// TwinCAT 3 PLC project motion
// Title: LCLS_OMotion
// Company: SLAC
// ProjectVersion: 6.0.0
// ProgramVersion: 3.1.4026.17
// libraries:
//   LCLS General, * (SLAC)
//   Tc2_EtherCAT, * (Beckhoff Automation GmbH)
//   Tc2_MC2, * (Beckhoff Automation GmbH)
//   Tc2_Standard, * (Beckhoff Automation GmbH)
//   Tc2_System, * (Beckhoff Automation GmbH)
//   Tc2_Utilities, * (Beckhoff Automation GmbH)
//   TcUnit, * (www.tcunit.org)
// project tree:
//   / DemoTask.TcTTO (not stored), PlcTask.TcTTO, UnitTestTask.TcTTO
//   DUTs/ E_LCLSMotionError.TcDUT, E_MotionLogLevel.TcDUT (not stored), MOTION_LOGGER_MSG.TcDUT (not stored), ST_ExtendedMotionStatus.TcDUT, E_HomeStates.TcDUT (not stored), E_Module.TcDUT (not stored), ST_MotionStatus.TcDUT, ENUM_StageEnableMode.TcDUT (not stored), E_DS402HomingMethod.TcDUT (not stored), E_DS402OpMode.TcDUT (not stored), E_EpicsHomeCmd.TcDUT, E_EpicsMotorCmd.TcDUT (not stored), E_MoveMode.TcDUT (not stored), E_MoveState.TcDUT, E_StageBrakeMode.TcDUT (not stored), E_StageEnableMode.TcDUT (not stored), ST_AxisParameterSetExposed.TcDUT (not stored), ST_DS402Drive.TcDUT, ST_DS402DriveStatus.TcDUT (not stored), ST_AxisStatus.TcDUT, ST_MotionCommand.TcDUT, ST_MotionLogMessage.TcDUT (not stored), ST_MoveRequestStatus.TcDUT
//   POUs/FBs/Common/ FB_EncoderScaling.TcPOU (not stored), FB_EpicsMotionParamsStatus.TcPOU (not stored), FB_EpicsMoveRequest.TcPOU (not stored), FB_LimSwStatus.TcPOU, FB_MotionDrive.TcPOU, FB_MotionDriveStateMachine.TcPOU (not stored), FB_MotionInterlocksCommon.TcPOU, FB_MotionInterlocksLimSw.TcPOU (not stored), FB_MotionLogger.TcPOU (not stored), FB_PersistentDataStorage.TcPOU (not stored)
//   POUs/FBs/Containers/ FB_MotionStageNC.TcPOU (not stored)
//   POUs/FBs/DS402/ FB_HomeDS402.TcPOU (excluded from build)
//   POUs/FBs/NC/ FB_AxisStatusNC.TcPOU (excluded from build), FB_BacklashCompensationNC.TcPOU, FB_BrakeNC.TcPOU, FB_HaltNC.TcPOU, FB_HomeNC.TcPOU, FB_MotionAxisNC.TcPOU, FB_MoveAbsoluteNC.TcPOU, FB_ParamsSaveRestoreNC.TcPOU, FB_PowerInterlockNC.TcPOU (not stored), FB_PowerNC.TcPOU, FB_ReadParameterNC.TcPOU, FB_ResetNC.TcPOU, FB_WriteParameterNC.TcPOU
//   POUs/ITFs/ I_AxisStatus.TcIO, I_BacklashCompensation.TcIO, I_Brake.TcIO, I_DS402GenericDrive.TcIO (not stored), I_EncoderScaling.TcIO (not stored), I_EpicsMotionParamsStatus.TcIO (not stored), I_Error.TcIO (not stored), I_Halt.TcIO, I_Home.TcIO, I_HomeDS402.TcIO (not stored), I_LimSwStatus.TcIO, I_MotionAxis.TcIO, I_MotionAxisDS402.TcIO, I_MotionDrive.TcIO, I_MotionInterlocks.TcIO, I_MotionInterlocksCommon.TcIO (not stored), I_MotionLogger.TcIO (not stored), I_MotionStage.TcIO (not stored), I_MoveAbsolute.TcIO, I_MoveRequest.TcIO (not stored), I_ParamsSaveRestore.TcIO (not stored), I_PersistentDataStorage.TcIO (not stored), I_Power.TcIO, I_ReadParameter.TcIO, I_Reset.TcIO, I_StateMachine.TcIO (not stored), I_Status.TcIO (not stored), I_StatusEx.TcIO (not stored), I_WriteParameter.TcIO (not stored)
//   Test/Containers/ FB_MotionStageNC_Test.TcPOU
//   Test/Interlok/ FB_MotionInterlocksCommon_Test.TcPOU, FB_MotionInterlocksLimSw_Test.TcPOU
//   Test/ HARD_TEST.TcPOU, PRG_TEST.TcPOU, CONTAINER_TEST.TcPOU
//   Test/Orchetration/ FB_BrakeNC_Test.TcPOU (not stored), FB_MotionDriveStateMachine_Test.TcPOU, FB_MotionDrive_Test.TcPOU, FB_MoveRequest_Test.TcPOU
//   Test/NC/ FB_NcMotionBlocks_Test.TcPOU, FB_MotionAxisNC_Test.TcPOU
//   Test/TestDouble/ FB_AxisStatusNC_TestDouble.TcPOU, FB_BacklashCompensationNC_TestDouble.TcPOU, FB_Brake_TestDouble.TcPOU (not stored), FB_EncoderScalingNC_TestDouble.TcPOU (not stored), FB_EpicsMotionParamsStatus_TestDouble.TcPOU, FB_HaltNC_TestDouble.TcPOU, FB_HomeNC_TestDouble.TcPOU, FB_LimSwStatus_testDouble.TcPOU, FB_MotionAxisDS402_TestDouble.TcPOU, FB_MotionAxisNC_TestDouble.TcPOU, FB_StateMachine_TestDouble.TcPOU, FB_MotionInterlocksCommon_TestDouble.TcPOU, FB_MotionInterlocksLimSw_TestDouble.TcPOU, FB_MotionLogger_TestDouble.TcPOU, FB_MoveAbsoluteNC_TestDouble.TcPOU, FB_MoveRequest_TestDouble.TcPOU, FB_ParamSaveRestoreNC_TestDouble.TcPOU (not stored), FB_PersistentDataStorage_TestDouble.TcPOU (not stored), FB_PowerNC_TestDouble.TcPOU, FB_ReadParameterNC_TestDouble.TcPOU (not stored), FB_ResetNC_TestDouble.TcPOU, FB_WriteParameterNC_TestDouble.TcPOU
//   Test/Utils/ FB_MotionLogger_Test.TcPOU
//   VISUs/ motion.TcCD (not stored)
// real-time tasks:
//   TASK PlcTask: cycle T#10ms, priority 1, ADS port 350
//   TASK UnitTestTask: cycle T#10ms, priority 20, ADS port 351
//   TASK Demo: cycle T#10ms, priority 2, ADS port 352
// motion (NC):
//   TASK NC-Task 1 SAF: cycle T#2ms, priority 4, ADS port 501
//   TASK NC-Task 1 SVB: cycle T#10ms, priority 8, ADS port 511
//   AXIS Axis_HomeNC_Test8 (id 15)
//     OtherSettings: AllowMotionCmdToSlave=true
//     encoder EncType=1
//     drive DrvType=5
//       Analog: TorqueSetpointScale=10, ScaleFactorActTorque=0.1
//       TimeComp: TaskDelayCycles=1
//     controller CtrType=1
//       CtrPara: PriorControlFactor=1
//         Observer: BandWidth=20
//   AXIS Axis_HomeNC_Test7 (id 14)
//     OtherSettings: AllowMotionCmdToSlave=true
//     encoder EncType=1
//     drive DrvType=5
//       Analog: TorqueSetpointScale=10, ScaleFactorActTorque=0.1
//       TimeComp: TaskDelayCycles=1
//     controller CtrType=1
//       CtrPara: PriorControlFactor=1
//         Observer: BandWidth=20
//   AXIS Axis_HomeNC_Test6 (id 2)
//     OtherSettings: AllowMotionCmdToSlave=true
//     encoder EncType=1
//     drive DrvType=5
//       Analog: TorqueSetpointScale=10, ScaleFactorActTorque=0.1
//       TimeComp: TaskDelayCycles=1
//     controller CtrType=1
//       CtrPara: PriorControlFactor=1
//         Observer: BandWidth=20
//   AXIS Axis_HomeNC_Test5 (id 7)
//     OtherSettings: AllowMotionCmdToSlave=true
//     encoder EncType=1
//     drive DrvType=5
//       Analog: TorqueSetpointScale=10, ScaleFactorActTorque=0.1
//       TimeComp: TaskDelayCycles=1
//     controller CtrType=1
//       CtrPara: PriorControlFactor=1
//         Observer: BandWidth=20
//   AXIS Axis_HomeNC_Test4 (id 6)
//     OtherSettings: AllowMotionCmdToSlave=true
//     encoder EncType=1
//     drive DrvType=5
//       Analog: TorqueSetpointScale=10, ScaleFactorActTorque=0.1
//       TimeComp: TaskDelayCycles=1
//     controller CtrType=1
//       CtrPara: PriorControlFactor=1
//         Observer: BandWidth=20
//   AXIS Axis_HomeNC_Test3 (id 5)
//     OtherSettings: AllowMotionCmdToSlave=true
//     encoder EncType=1
//     drive DrvType=5
//       Analog: TorqueSetpointScale=10, ScaleFactorActTorque=0.1
//       TimeComp: TaskDelayCycles=1
//     controller CtrType=1
//       CtrPara: PriorControlFactor=1
//         Observer: BandWidth=20
//   AXIS Axis_HomeNC_Test2 (id 4)
//     Velo: RefSearch=500, RefSync=500
//     OtherSettings: AllowMotionCmdToSlave=true
//     encoder EncType=1
//     drive DrvType=5
//       Analog: TorqueSetpointScale=10, ScaleFactorActTorque=0.1
//       TimeComp: TaskDelayCycles=1
//     controller CtrType=1
//       CtrPara: PriorControlFactor=1
//         Observer: BandWidth=20
//   AXIS Axis_HomeNC_Test1 (id 3)
//     OtherSettings: AllowMotionCmdToSlave=true
//     encoder EncType=1
//     drive DrvType=5
//       Analog: TorqueSetpointScale=10, ScaleFactorActTorque=0.1
//       TimeComp: TaskDelayCycles=1
//     controller CtrType=1
//       CtrPara: PriorControlFactor=1
//         Observer: BandWidth=20
//   AXIS Axis_McMotionBlocks_Test1 (id 9)
//     OtherSettings: AllowMotionCmdToSlave=true
//     encoder EncType=1
//     drive DrvType=5
//       Analog: TorqueSetpointScale=10, ScaleFactorActTorque=0.1
//       TimeComp: TaskDelayCycles=1
//     controller CtrType=1
//       CtrPara: PriorControlFactor=1
//         Observer: BandWidth=20
//   AXIS Axis_McMotionBlocks_Test2 (id 10)
//     OtherSettings: AllowMotionCmdToSlave=true
//     encoder EncType=1
//     drive DrvType=5
//       Analog: TorqueSetpointScale=10, ScaleFactorActTorque=0.1
//       TimeComp: TaskDelayCycles=1
//     controller CtrType=1
//       CtrPara: PriorControlFactor=1
//         Observer: BandWidth=20
//   AXIS Axis_McMotionBlocks_Test3 (id 11)
//     OtherSettings: AllowMotionCmdToSlave=true
//     encoder EncType=1
//     drive DrvType=5
//       Analog: TorqueSetpointScale=10, ScaleFactorActTorque=0.1
//       TimeComp: TaskDelayCycles=1
//     controller CtrType=1
//       CtrPara: PriorControlFactor=1
//         Observer: BandWidth=20
//   AXIS Axis_McMotionBlocks_Test4 (id 12)
//     OtherSettings: AllowMotionCmdToSlave=true
//     encoder EncType=1
//     drive DrvType=5
//       Analog: TorqueSetpointScale=10, ScaleFactorActTorque=0.1
//       TimeComp: TaskDelayCycles=1
//     controller CtrType=1
//       CtrPara: PriorControlFactor=1
//         Observer: BandWidth=20
//   AXIS Axis_McMotionBlocks_Test8 (id 17)
//     OtherSettings: AllowMotionCmdToSlave=true
//     encoder EncType=1
//       ActPosCorrection: Enable=true
//     drive DrvType=5
//       Analog: TorqueSetpointScale=10, ScaleFactorActTorque=0.1
//       TimeComp: TaskDelayCycles=1
//     controller CtrType=1
//       CtrPara: PriorControlFactor=1
//         Observer: BandWidth=20
//   AXIS Axis_McMotionBlocks_Test7 (id 1)
//     OtherSettings: AllowMotionCmdToSlave=true
//     encoder EncType=1
//       ActPosCorrection: Enable=true
//     drive DrvType=5
//       Analog: TorqueSetpointScale=10, ScaleFactorActTorque=0.1
//       TimeComp: TaskDelayCycles=1
//     controller CtrType=1
//       CtrPara: PriorControlFactor=1
//         Observer: BandWidth=20
//   AXIS Axis_McMotionBlocks_Test6 (id 16)
//     OtherSettings: AllowMotionCmdToSlave=true
//     encoder EncType=1
//       ActPosCorrection: Enable=true
//     drive DrvType=5
//       Analog: TorqueSetpointScale=10, ScaleFactorActTorque=0.1
//       TimeComp: TaskDelayCycles=1
//     controller CtrType=1
//       CtrPara: PriorControlFactor=1
//         Observer: BandWidth=20
//   AXIS Axis_McMotionBlocks_Test5 (id 13)
//     OtherSettings: AllowMotionCmdToSlave=true
//     encoder EncType=1
//     drive DrvType=5
//       Analog: TorqueSetpointScale=10, ScaleFactorActTorque=0.1
//       TimeComp: TaskDelayCycles=1
//     controller CtrType=1
//       CtrPara: PriorControlFactor=1
//         Observer: BandWidth=20
//   AXIS Axis_Hard_Test (id 8)
//     Velo: RefSync=100
//     OtherSettings: AllowMotionCmdToSlave=true
//     encoder EncType=1
//       ActPosCorrection: Enable=true
//     drive DrvType=5
//       Analog: TorqueSetpointScale=10, ScaleFactorActTorque=0.1
//       TimeComp: TaskDelayCycles=1
//     controller CtrType=1
//       CtrPara: PriorControlFactor=1
//         Observer: BandWidth=20
// variable links:
//   motion/motion Instance <-> NC-Task 1 SAF/Axes/Axis_Hard_Test
//     DemoTask Inputs/NcAxis_GVL.NC.NcToPlc <-> Outputs/ToPlc
//     DemoTask Outputs/NcAxis_GVL.NC.PlcToNc <-> Inputs/FromPlc
//   motion/motion Instance <-> NC-Task 1 SAF/Axes/Axis_HomeNC_Test1
//     UnitTestTask Inputs/PRG_TEST.fb_HomeNC_Test.fbAxisRef[1].NcToPlc <-> Outputs/ToPlc
//     UnitTestTask Outputs/PRG_TEST.fb_HomeNC_Test.fbAxisRef[1].PlcToNc <-> Inputs/FromPlc
//   motion/motion Instance <-> NC-Task 1 SAF/Axes/Axis_HomeNC_Test2
//     UnitTestTask Inputs/PRG_TEST.fb_HomeNC_Test.fbAxisRef[2].NcToPlc <-> Outputs/ToPlc
//     UnitTestTask Outputs/PRG_TEST.fb_HomeNC_Test.fbAxisRef[2].PlcToNc <-> Inputs/FromPlc
//   motion/motion Instance <-> NC-Task 1 SAF/Axes/Axis_HomeNC_Test3
//     UnitTestTask Inputs/PRG_TEST.fb_HomeNC_Test.fbAxisRef[3].NcToPlc <-> Outputs/ToPlc
//     UnitTestTask Outputs/PRG_TEST.fb_HomeNC_Test.fbAxisRef[3].PlcToNc <-> Inputs/FromPlc
//   motion/motion Instance <-> NC-Task 1 SAF/Axes/Axis_HomeNC_Test4
//     UnitTestTask Inputs/PRG_TEST.fb_HomeNC_Test.fbAxisRef[4].NcToPlc <-> Outputs/ToPlc
//     UnitTestTask Outputs/PRG_TEST.fb_HomeNC_Test.fbAxisRef[4].PlcToNc <-> Inputs/FromPlc
//   motion/motion Instance <-> NC-Task 1 SAF/Axes/Axis_HomeNC_Test5
//     UnitTestTask Inputs/PRG_TEST.fb_HomeNC_Test.fbAxisRef[5].NcToPlc <-> Outputs/ToPlc
//     UnitTestTask Outputs/PRG_TEST.fb_HomeNC_Test.fbAxisRef[5].PlcToNc <-> Inputs/FromPlc
//   motion/motion Instance <-> NC-Task 1 SAF/Axes/Axis_HomeNC_Test6
//     UnitTestTask Inputs/PRG_TEST.fb_HomeNC_Test.fbAxisRef[6].NcToPlc <-> Outputs/ToPlc
//     UnitTestTask Outputs/PRG_TEST.fb_HomeNC_Test.fbAxisRef[6].PlcToNc <-> Inputs/FromPlc
//   motion/motion Instance <-> NC-Task 1 SAF/Axes/Axis_HomeNC_Test7
//     UnitTestTask Inputs/PRG_TEST.fb_HomeNC_Test.fbAxisRef[7].NcToPlc <-> Outputs/ToPlc
//     UnitTestTask Outputs/PRG_TEST.fb_HomeNC_Test.fbAxisRef[7].PlcToNc <-> Inputs/FromPlc
//   motion/motion Instance <-> NC-Task 1 SAF/Axes/Axis_HomeNC_Test8
//     UnitTestTask Inputs/PRG_TEST.fb_HomeNC_Test.fbAxisRef[8].NcToPlc <-> Outputs/ToPlc
//     UnitTestTask Outputs/PRG_TEST.fb_HomeNC_Test.fbAxisRef[8].PlcToNc <-> Inputs/FromPlc
//   motion/motion Instance <-> NC-Task 1 SAF/Axes/Axis_McMotionBlocks_Test1
//     UnitTestTask Inputs/PRG_TEST.fb_McMotionBlocks_Test.fbAxisRef[1].NcToPlc <-> Outputs/ToPlc
//     UnitTestTask Outputs/PRG_TEST.fb_McMotionBlocks_Test.fbAxisRef[1].PlcToNc <-> Inputs/FromPlc
//   motion/motion Instance <-> NC-Task 1 SAF/Axes/Axis_McMotionBlocks_Test2
//     UnitTestTask Inputs/PRG_TEST.fb_McMotionBlocks_Test.fbAxisRef[2].NcToPlc <-> Outputs/ToPlc
//     UnitTestTask Outputs/PRG_TEST.fb_McMotionBlocks_Test.fbAxisRef[2].PlcToNc <-> Inputs/FromPlc
//   motion/motion Instance <-> NC-Task 1 SAF/Axes/Axis_McMotionBlocks_Test3
//     UnitTestTask Inputs/PRG_TEST.fb_McMotionBlocks_Test.fbAxisRef[3].NcToPlc <-> Outputs/ToPlc
//     UnitTestTask Outputs/PRG_TEST.fb_McMotionBlocks_Test.fbAxisRef[3].PlcToNc <-> Inputs/FromPlc
//   motion/motion Instance <-> NC-Task 1 SAF/Axes/Axis_McMotionBlocks_Test4
//     UnitTestTask Inputs/PRG_TEST.fb_McMotionBlocks_Test.fbAxisRef[4].NcToPlc <-> Outputs/ToPlc
//     UnitTestTask Outputs/PRG_TEST.fb_McMotionBlocks_Test.fbAxisRef[4].PlcToNc <-> Inputs/FromPlc
//   motion/motion Instance <-> NC-Task 1 SAF/Axes/Axis_McMotionBlocks_Test5
//     UnitTestTask Inputs/PRG_TEST.fb_McMotionBlocks_Test.fbAxisRef[5].NcToPlc <-> Outputs/ToPlc
//     UnitTestTask Outputs/PRG_TEST.fb_McMotionBlocks_Test.fbAxisRef[5].PlcToNc <-> Inputs/FromPlc
//   motion/motion Instance <-> NC-Task 1 SAF/Axes/Axis_McMotionBlocks_Test6
//     UnitTestTask Inputs/PRG_TEST.fb_McMotionBlocks_Test.fbAxisRef[6].NcToPlc <-> Outputs/ToPlc
//     UnitTestTask Outputs/PRG_TEST.fb_McMotionBlocks_Test.fbAxisRef[6].PlcToNc <-> Inputs/FromPlc
//   motion/motion Instance <-> NC-Task 1 SAF/Axes/Axis_McMotionBlocks_Test7
//     UnitTestTask Inputs/PRG_TEST.fb_McMotionBlocks_Test.fbAxisRef[7].NcToPlc <-> Outputs/ToPlc
//     UnitTestTask Outputs/PRG_TEST.fb_McMotionBlocks_Test.fbAxisRef[7].PlcToNc <-> Inputs/FromPlc
//   motion/motion Instance <-> NC-Task 1 SAF/Axes/Axis_McMotionBlocks_Test8
//     UnitTestTask Inputs/PRG_TEST.fb_McMotionBlocks_Test.fbAxisRef[8].NcToPlc <-> Outputs/ToPlc
//     UnitTestTask Outputs/PRG_TEST.fb_McMotionBlocks_Test.fbAxisRef[8].PlcToNc <-> Inputs/FromPlc

CONFIGURATION motion
    RESOURCE PLC ON TwinCAT3
        TASK PlcTask(INTERVAL := T#10ms, PRIORITY := 1);
        TASK UnitTestTask(INTERVAL := T#10ms, PRIORITY := 20);
        PROGRAM MAIN WITH PlcTask : MAIN;
        PROGRAM PRG_TEST WITH UnitTestTask : PRG_TEST;
    END_RESOURCE
END_CONFIGURATION

// ---- DUTs/E_LCLSMotionError.TcDUT
{attribute 'qualified_only'}
{attribute 'strict'}
{attribute 'to_string'}
TYPE E_LCLSMotionError :
(
    ABORTED := 16#7900,
    UNSAFE := 16#7901,
    INVALID := 16#7902,
    TEST := 16#FFFF
)UDINT;
END_TYPE

// ---- DUTs/ST_ExtendedMotionStatus.TcDUT
TYPE ST_ExtendedMotionStatus :
STRUCT
	bMotionAxisError : BOOL;
	nMotionAxisErrorId : UDINT;
	bInterlocksError : BOOL;
	nInterlocksError : UDINT;
	eDriveState : E_MoveState;
	bDriveWatchDogStatus : BOOL;
	bAbortDone : BOOL;
	bAborted : BOOL;
	bLimHomeDone : BOOL;
	bNewMoveReq : BOOL;
	bEnable : BOOL;
	bIdling : BOOL;
END_STRUCT
END_TYPE

// ---- DUTs/ST_MotionStatus.TcDUT
TYPE ST_MotionStatus :
STRUCT
   {attribute 'pytmc' := '
        pv: PLC:bLimitFwd
        io: i
        field: DESC Error code if nonzero
    '}
	bLimitFwd: BOOL;

    {attribute 'pytmc' := '
        pv: PLC:bLimitBwd
        io: i
        field: DESC Error code if nonzero
    '}
	bLimitBwd: BOOL;

    {attribute 'pytmc' := '
        pv: PLC:bHomeSensor
        io: i
        field: DESC Error code if nonzero
    '}
	bHomeSensor: BOOL;

    {attribute 'pytmc' := '
        pv: PLC:bEnabled
        io: i
        field: DESC Error code if nonzero
        update: 100Hz notify
    '}
	bEnabled: BOOL;

    // Used internally and by the IOC to pick a destination for the move
    {attribute 'pytmc' := '
        pv: PLC:fOverride
        io: i
        field: DESC Used internally to set power override
    '}
	fOverride : LREAL;

    {attribute 'pytmc' := '
        pv: PLC:fActVelocity
        io: i
        field: DESC Error code if nonzero
    '}
	fActVelocity: LREAL;

    {attribute 'pytmc' := '
        pv: PLC:fActPosition
        io: i
        field: DESC Error code if nonzero
    '}
	fActPosition: LREAL;

    {attribute 'pytmc' := '
        pv: PLC:fActDiff
        io: i
        field: DESC Error code if nonzero
        update: 100Hz notify
    '}
	fActDiff: LREAL;

    // TRUE if in the middle of a command
    {attribute 'pytmc' := '
        pv: PLC:bBusy
        io: i
        field: ZNAM FALSE
        field: ONAM TRUE
        field: DESC TRUE if in the middle of a command
        update: 100Hz notify
    '}
    bBusy: BOOL;

    // TRUE if we've done a command and it has finished
    {attribute 'pytmc' := '
        pv: PLC:bDone
        io: i
        field: ZNAM FALSE
        field: ONAM TRUE
        field: DESC TRUE if we've done a command AND it has finished
        update: 100Hz notify
    '}
    bDone: BOOL;

    // TRUE if the motor has been homed, or does not need to be homed
    {attribute 'pytmc' := '
        pv: PLC:bHomed
        io: i
        field: ZNAM FALSE
        field: ONAM TRUE
        field: DESC TRUE if the motor has been homed, or does not need to be homed
        update: 100Hz notify
    '}
    bHomed: BOOL;
	
    {attribute 'pytmc' := '
        pv: PLC:bWarning
        io: i
        field: ZNAM FALSE
        field: ONAM TRUE
        field: DESC Interlocks Warning
    '}	
	bWarning : BOOL;
	
    // TRUE if we're in an error state
    {attribute 'pytmc' := '
        pv: PLC:bError
        io: i
        field: ZNAM FALSE
        field: ONAM TRUE
        field: DESC TRUE if we are in an error state
        update: 100Hz notify
    '}
    bError: BOOL;

    // Error code if nonzero
    {attribute 'pytmc' := '
        pv: PLC:nErrorId
        io: i
        field: DESC Error code if nonzero
        update: 100Hz notify
    '}
    nErrorId: UDINT;

    // Unique ID assigned to each axis in the NC
    {attribute 'pytmc' := '
        pv: PLC:nMotionAxisID
        io: i
        field: DESC Unique ID assigned to each axis in the NC
    '}
    nMotionAxisID: UDINT:=0;

    // Message to identify the error state
    {attribute 'pytmc' := '
        pv: PLC:sErrorMessage
        io: i
        field: DESC Message to identify the error state
        update: 100Hz notify
    '}
    sErrorMessage: STRING;
END_STRUCT
END_TYPE

// ---- DUTs/E_EpicsHomeCmd.TcDUT
{attribute 'qualified_only'}
{attribute 'strict'}
TYPE E_EpicsHomeCmd :
    // Defines the valid options for homing in FB_MotionStage
(
    LOW_LIMIT := 1, // Low limit switch
    HIGH_LIMIT := 2, // High limit switch
    HOME_VIA_LOW := 3, // Home switch via low switch
    HOME_VIA_HIGH := 4, // Home switch via high switch
    ABSOLUTE_SET := 15, // Set here to be fHomePosition
    // MCS2
    AUTOZERO := -1,
    CURRENT_POSITION_METHOD := 37,
    NONE := -99 // Do not home, ever
) := NONE;
END_TYPE

// ---- DUTs/E_MoveState.TcDUT
{attribute 'qualified_only'}
{attribute 'strict'}
{attribute 'to_string'}
TYPE E_MoveState :
(
    IDLING:=0,
    INIT:=10,
    STARTED:=20,
    IN_PROGRESS :=30,
    REACHED:=40,
    INTERRUPTED:=50,
    DONE:=60,
    ERROR:=-99
);
END_TYPE

// ---- DUTs/ST_DS402Drive.TcDUT
TYPE ST_DS402Drive:
STRUCT
    (* Global variables for the TPDO data from the drive. Each one is linked to the respective TPDO channel. *)
    stDriveStatus 			AT %I*	: 	ST_DS402DriveStatus;
    nModeOfOperationDisplay AT %I*	: 	SINT;
    //nActualPosition 		AT %I*	: 	DINT;
    (*CSP drive mode*)
    nFollowingError 		AT %I*	: 	DINT;
    (* Global variables for the RPDO data to the drive. Each one is linked to the respective RPDO channel. *)
    //nDS402DriveControl		AT %Q*	:	UINT;
	// Connected to NC task Ctrl 1 and Ctrl 2
   	nDS402DriveControlNC	AT %I*	:	UINT;
	// connected to I/O Task 'Control Word'
   	nDS402DriveControl		AT %Q*	:	UINT;
    //nTargetPositionTmp 		AT %I* 	: 	DINT;
    nTargetPosition 		AT %Q* 	: 	DINT;
    nModeOfOperationNC 	AT %I* 	: 	SINT;
    nModeOfOperation 		AT %Q* 	: 	SINT;
    (* Global variables for the RPDO data to the drive. Each one is linked to the respective RPDO channel. *)
    nProfilVelocity 		AT %Q* 	: 	DINT;
    nProfilAcceleration		AT %Q* 	: 	DINT;
    nProfilDecceleration	AT %Q* 	: 	DINT;
    nVelocityActualValue	AT %Q* 	: 	DINT;
    (* Global variables for the TPDO data from the drive. Each one is linked to the respective TPDO channel. *)
    nScantargetPosition		AT %Q*	: 	DINT;
    uScantargetVelocity		AT %Q*	: 	ULINT;

    {attribute 'pytmc' := '
        pv: PLC:nChanStep
        io: io
        field: DESC SmartAct: Open Loop Step Count
    '}
    nChanStep			: DINT;

    {attribute 'pytmc' := '
        pv: PLC:nChanStepFreq
        io: io
        field: DESC SmartAct: Open Loop Step Freq
    '}
    nChanStepFreq		: UINT;

    {attribute 'pytmc' := '
        pv: PLC:nChanStepAmp
        io: io
        field: DESC SmartAct: Open Loop Step Amp
    '}
    nChanStepAmp		: UINT;

    // timeout for holding actual position in close loop mode
    {attribute 'pytmc' := '
        pv: PLC:nHoldTime
        io: io
        field: DESC SmartAct: Set servo mode hold time
    '}
    nHoldTime						: UDINT := 10000;

    {attribute 'pytmc' := '
        pv: PLC:bServo
        io: io
        field: ZNAM DISABLE
        field: ONAM ENABLE
        field: DESC Used to disable close loop mode
    '}
    bServo							: BOOL := TRUE;

    (* NetId of EtherCAT Master *)
    arNetId  				AT %I*	: 	AMSNETID;
    (* Port Number of EtherCAT Slave *)
    nSlaveAddr 				AT %I* 	: 	UINT;

END_STRUCT
END_TYPE

// ---- DUTs/ST_AxisStatus.TcDUT
TYPE ST_AxisStatus :
STRUCT
	nAxisId : UDINT;
	bAxisEnable : BOOL;
	bAbortDone : BOOL;
	bAborted : BOOL;
	bAxisReadParamsInit : BOOL;
	eAxisState : MC_AxisStates;
	bBacklashCompensationStatus : BOOL;
	bBusy : BOOL;
	bDone : BOOL;
	bError : BOOL;
	nErrorID : UDINT;
	bHaltActive : BOOL;
	bHaltBusy : BOOL;
	bHaltDone : BOOL;
	bHomeBusy : BOOL;
	bHomeDone : BOOL;
	bLimHomeDone : BOOL;
	nHomeMode : INT;
	bInTargetPosition : BOOL;
	fMeasuredAcceleration : LREAL;
	fMeasuredCompensation : LREAL;
	fMeasuredPosition : LREAL;
	fMeasuredPositionDiff : LREAL;
	fMeasuredVelocity : LREAL;
	sMessage : T_MaxString;
	bMoveAbsoluteAborted : BOOL;
	bMoveAbsoluteActive : BOOL;
	bMoveAbsoluteBusy : BOOL;
	bMoveAbsoluteDone : BOOL;
	bNegativeMotionIsEnabled : BOOL;
	bPositiveMotionIsEnabled : BOOL;
	bDirectionalPowerEnabled : BOOL;
	bPowerActive : BOOL;
	bPowerIsEnabled : BOOL;
	fPowerOverride : LREAL;
	bResetBusy : BOOL;
	bResetDone : BOOL;
	bRestoreDone : BOOL;
	fSavedPosition : LREAL;
	nScaledEncoderCount : UDINT;
	bStandStill : BOOL;
END_STRUCT
END_TYPE

// ---- DUTs/ST_MotionCommand.TcDUT
TYPE ST_MotionCommand :
    // Defines the EPICS interface to moving a motor in TwinCAT
STRUCT
    // Used internally to reset errors and other state
    {attribute 'pytmc' := '
        pv: PLC:bReset
        io: io
        field: ZNAM FALSE
        field: ONAM TRUE
        field: DESC Used internally to reset errors
    '}
    bReset: BOOL;
    {attribute 'pytmc' := '
        pv: PLC:bHalt
        io: io
        field: ZNAM FALSE
        field: ONAM TRUE
        field: DESC Used internally to stop move
    '}
    bHalt: BOOL;
    // Used internally and by the IOC to start or stop a move
    {attribute 'pytmc' := '
        pv: PLC:bMoveCmd
        io: io
        field: DESC Start an AbsoluteMove
    '}
    bMoveCmd	: BOOL;
    // Start the homing routine
    {attribute 'pytmc' := '
        pv: PLC:bHomeCmd
        io: io
        field: DESC Start the homing routine
    '}
    bHomeCmd: BOOL;
	
    //bExecute: BOOL;
    // Used internally and by the IOC to pick what kind of move to do
    {attribute 'pytmc' := '
        pv: PLC:nCommand
        io: io
        field: DESC Used internally and by the IOC to pick what kind of move to do
    '}
	nCommand: INT;
    // Used internally and by the IOC to pass additional data to some commands
    {attribute 'pytmc' := '
        pv: PLC:nCmdData
        io: io
        field: DESC Used internally and by the IOC to pass additional data to some commands
    '}
	nCmdData: INT;	

    // Used internally and by the IOC to pick a destination for the move
    {attribute 'pytmc' := '
        pv: PLC:fPosition
        io: io
        field: DESC Used internally and by the IOC to pick a destination for the move
    '}
    fPosition: LREAL;

    // Used internally and by the IOC to pick a move velocity
    {attribute 'pytmc' := '
        pv: PLC:fVelocity
        io: io
        field: DESC Used internally and by the IOC to pick a move velocity
    '}
    fVelocity: LREAL;

    // Used internally and by the IOC to pick a move acceleration
    {attribute 'pytmc' := '
        pv: PLC:fAcceleration
        io: io
        field: DESC Used internally and by the IOC to pick a move acceleration
    '}
    fAcceleration: LREAL;

    // Used internally and by the IOC to pick a move deceleration
    {attribute 'pytmc' := '
        pv: PLC:fDeceleration
        io: io
        field: DESC Used internally and by the IOC to pick a move deceleration
    '}
    fDeceleration: LREAL;

    // Used internally and by the IOC to pick a move jerk
    {attribute 'pytmc' := '
        pv: PLC:fJerk
        io: io
        field: DESC Used internally and by the IOC to pick a move jerk
    '}
    fJerk: LREAL;

    // Used internally and by the IOC to pick a home position
    {attribute 'pytmc' := '
        pv: PLC:fHomePosition
        io: io
        field: DESC Used internally and by the IOC to pick home position
    '}
    fHomePosition: LREAL;

END_STRUCT
END_TYPE

// ---- DUTs/ST_MoveRequestStatus.TcDUT
TYPE ST_MoveRequestStatus :
STRUCT
    bEnable: BOOL;
    bNewMoveReq: BOOL;
	bExecute: BOOL;
    nCmdData: INT;
    nCommand: INT;
    bExecHome: BOOL;
	bHomeEnablewOverride : BOOL;
    bExecMove: BOOL;
	bPrepareDisable : BOOL;
END_STRUCT
END_TYPE

// ---- POUs/ITFs/I_AxisStatus.TcIO
INTERFACE I_AxisStatus EXTENDS I_Output

METHOD AxisEnabled : BOOL
VAR_INPUT
END_VAR
END_METHOD

PROPERTY AxisID : UDINT
GET
END_GET
END_PROPERTY

PROPERTY AxisState : MC_AxisStates
GET
END_GET
END_PROPERTY

PROPERTY InTargetPosition : BOOL
GET
END_GET
END_PROPERTY

PROPERTY MeasuredAcceleration : LREAL
GET
END_GET
END_PROPERTY

PROPERTY MeasuredPosition : LREAL
GET
END_GET
END_PROPERTY

PROPERTY MeasuredPositionDiff : LREAL
GET
END_GET
END_PROPERTY

PROPERTY MeasuredVelocity : LREAL
GET
END_GET
END_PROPERTY

PROPERTY NegativeMotionIsEnabled : BOOL
GET
END_GET
END_PROPERTY

PROPERTY PositiveMotionIsEnabled : BOOL
GET
END_GET
END_PROPERTY

PROPERTY StandStill : BOOL
GET
END_GET
END_PROPERTY

PROPERTY Stopped : BOOL
GET
END_GET
END_PROPERTY

END_INTERFACE

// ---- POUs/ITFs/I_BacklashCompensation.TcIO
INTERFACE I_BacklashCompensation EXTENDS I_Error

METHOD BacklashCompensation
VAR_INPUT
	Enable : BOOL := FALSE;
	RampVelo : LREAL;
END_VAR
END_METHOD

PROPERTY Busy : BOOL
GET
END_GET
END_PROPERTY

METHOD ClearStatus
VAR_INPUT
END_VAR
END_METHOD

PROPERTY CurrentBacklash : LREAL
GET
END_GET
END_PROPERTY

METHOD EnableBacklashCompensation
VAR_INPUT
    UserEnable : BOOL;
    Compensation : LREAL;
END_VAR
END_METHOD

PROPERTY Status : BOOL
GET
END_GET
END_PROPERTY

END_INTERFACE

// ---- POUs/ITFs/I_Brake.TcIO
INTERFACE I_Brake EXTENDS I_Outputs

PROPERTY AxisState : MC_AxisStates
SET
END_SET
END_PROPERTY

PROPERTY BrakeMode : E_StageBrakeMode
GET
END_GET
SET
END_SET
END_PROPERTY

PROPERTY BrakeRelease : BOOL
GET
END_GET
END_PROPERTY

END_INTERFACE

// ---- POUs/ITFs/I_Halt.TcIO
INTERFACE I_Halt

METHOD Halt
VAR_INPUT
	Execute : BOOL;
    Deceleration : LREAL := 0.0;
    Jerk : LREAL := 0.0;
    BufferMode	: MC_BufferMode := MC_BufferMode.MC_Aborting;
END_VAR
END_METHOD

PROPERTY HaltActive : BOOL
GET
END_GET
END_PROPERTY

PROPERTY HaltBusy : BOOL
GET
END_GET
END_PROPERTY

PROPERTY HaltDone : BOOL
GET
END_GET
END_PROPERTY

PROPERTY HaltError : BOOL
GET
END_GET
END_PROPERTY

PROPERTY HaltErrorID : UDINT
GET
END_GET
END_PROPERTY

END_INTERFACE

// ---- POUs/ITFs/I_Home.TcIO
INTERFACE I_Home

PROPERTY CommandMoveHome : BOOL
SET
END_SET
END_PROPERTY

METHOD  Home
VAR_INPUT
	Execute	: BOOL;
	HomeSpeedFast	: LREAL;
	HomeSpeedSlow	: LREAL;
END_VAR
END_METHOD

PROPERTY HomeAbort : BOOL
GET
END_GET
SET
END_SET
END_PROPERTY

{warning 'add property implementation'}
PROPERTY HomeBusy : BOOL
GET
END_GET
END_PROPERTY

{warning 'add property implementation'}
PROPERTY HomeDone : BOOL
GET
END_GET
END_PROPERTY

{warning 'add property implementation'}
PROPERTY HomeError : BOOL
GET
END_GET
END_PROPERTY

{warning 'add property implementation'}
PROPERTY HomeErrorID : UDINT
GET
END_GET
END_PROPERTY

PROPERTY HomeMode : E_EpicsHomeCmd
GET
END_GET
SET
END_SET
END_PROPERTY

{warning 'Add property implementation'}
PROPERTY HomeOffset : LREAL
SET
END_SET
END_PROPERTY

{warning 'Add property implementation'}
PROPERTY HomePosition : LREAL
SET
END_SET
END_PROPERTY

END_INTERFACE

// ---- POUs/ITFs/I_LimSwStatus.TcIO
INTERFACE I_LimSwStatus

METHOD AxisStatus
VAR_INPUT
	HomeBusy: BOOL;
	PositiveDirection : BOOL;
	NegativeDirection : BOOL;
END_VAR
END_METHOD

METHOD DriveCommands
VAR_INPUT
	Enable: BOOL;
	NewMoveReq : BOOL;
	Reset: BOOL;
END_VAR
END_METHOD

PROPERTY LimBackward : BOOL
GET
END_GET
END_PROPERTY

PROPERTY LimForward : BOOL
GET
END_GET
END_PROPERTY

PROPERTY LimHit : BOOL
GET
END_GET
END_PROPERTY

PROPERTY LimHome : BOOL
GET
END_GET
END_PROPERTY

PROPERTY Message : T_MAXSTRING
GET
END_GET
END_PROPERTY

PROPERTY MoveBackwardEnabled : BOOL
GET
END_GET
END_PROPERTY

PROPERTY MoveForwardEnabled : BOOL
GET
END_GET
END_PROPERTY

PROPERTY Warning : BOOL
GET
END_GET
END_PROPERTY

END_INTERFACE

// ---- POUs/ITFs/I_MotionAxis.TcIO
INTERFACE I_MotionAxis EXTENDS __SYSTEM.IQueryInterface,

PROPERTY AbortDone : BOOL
GET
END_GET
END_PROPERTY

{warning 'Add property implementation'}
PROPERTY Aborted : BOOL
GET
END_GET
END_PROPERTY

METHOD AxisEnabled : BOOL
VAR_INPUT
	HomeCmd : BOOL;

	NewMoveReq : BOOL; 
END_VAR
END_METHOD

PROPERTY AxisReadParamsInit : BOOL
GET
END_GET
END_PROPERTY

PROPERTY AxisState : MC_AxisStates
GET
END_GET
END_PROPERTY

(*
    Handle positive/negative backlash compensation
    User needs to set the direction of backlash from the sign of the compensation value
    Backlash compensation is disabled during referencing (homing).
    When direction is positive/negative, further movement in the negative/positive direction not compensated
    further movement in the negative/positive direction will be compensated
*)
METHOD BacklashCompensation
VAR_INPUT
    Active     : BOOL;
    Compensation	: LREAL;
    RampVelocity	: LREAL;
    DisableMode	: E_DISABLEMODE := E_DISABLEMODE.DisableModeHold;
END_VAR
END_METHOD

(*synced Fbs need just to activate the compensation with a given ramp speed
  other parameters are provided via EPICS (declared in this FB) or via the more extended BackalshCompensation method (simulation) *)
METHOD BacklashCompensationActive
VAR_INPUT
    Active     : BOOL;
    RampVelocity : LREAL;
END_VAR
END_METHOD

{warning 'Add property implementation'}
PROPERTY BacklashCompStatus : BOOL
GET
END_GET
END_PROPERTY

PROPERTY BacklashCompUserEn : BOOL
SET
END_SET
END_PROPERTY

{warning 'add property implementation'}
PROPERTY Busy : BOOL
GET
END_GET
END_PROPERTY

{warning 'add property implementation'}
PROPERTY Done : BOOL
GET
END_GET
END_PROPERTY

{warning 'add property implementation'}
PROPERTY Error : BOOL
GET
END_GET
END_PROPERTY

{warning 'add property implementation'}
PROPERTY ErrorID : UDINT
GET
END_GET
END_PROPERTY

METHOD Halt
VAR_INPUT
	Execute : BOOL;
    Deceleration : LREAL := 0.0;
    Jerk : LREAL := 0.0;
    BufferMode	: MC_BufferMode := MC_BufferMode.MC_Aborting;
END_VAR
END_METHOD

{warning 'Add property implementation'}
PROPERTY HaltActive : BOOL
GET
END_GET
END_PROPERTY

PROPERTY HaltBusy : BOOL
GET
END_GET
END_PROPERTY

PROPERTY HaltDone : BOOL
GET
END_GET
END_PROPERTY

METHOD  Home
VAR_INPUT
	Execute	: BOOL;
	HomeSpeedFast	: LREAL;
	HomeSpeedSlow	: LREAL;
END_VAR
END_METHOD

PROPERTY HomeBusy : BOOL
GET
END_GET
END_PROPERTY

PROPERTY HomeDone : BOOL
GET
END_GET
END_PROPERTY

PROPERTY HomeMode : E_EpicsHomeCmd
GET
END_GET
END_PROPERTY

PROPERTY InTargetPosition : BOOL
GET
END_GET
END_PROPERTY

PROPERTY MeasuredAcceleration : LREAL
GET
END_GET
END_PROPERTY

{warning 'Add property implementation'}
PROPERTY MeasuredCompensation : LREAL
GET
END_GET
END_PROPERTY

PROPERTY MeasuredPosition : LREAL
GET
END_GET
END_PROPERTY

PROPERTY MeasuredPositionDiff : LREAL
GET
END_GET
END_PROPERTY

PROPERTY MeasuredVelocity : LREAL
GET
END_GET
END_PROPERTY

PROPERTY Message : T_MAXSTRING
GET
END_GET
END_PROPERTY

METHOD MoveAbsolute
VAR_INPUT
    Execute     : BOOL;
    Position	: LREAL;
    Velocity	: LREAL;
    Acceleration	: LREAL := 0.0;
    Deceleration	: LREAL := 0.0;
    Jerk	: LREAL := 0.0;
    BufferMode	: MC_BufferMode := MC_BufferMode.MC_Aborting;
END_VAR
END_METHOD

PROPERTY MoveAbsoluteAborted : BOOL
GET
END_GET
END_PROPERTY

PROPERTY MoveAbsoluteActive : BOOL
GET
END_GET
END_PROPERTY

PROPERTY MoveAbsoluteBusy : BOOL
GET
END_GET
END_PROPERTY

PROPERTY MoveAbsoluteDone : BOOL
GET
END_GET
END_PROPERTY

PROPERTY NegativeMotionIsEnabled : BOOL
GET
END_GET
END_PROPERTY

PROPERTY PositiveMotionIsEnabled : BOOL
GET
END_GET
END_PROPERTY

METHOD Power
VAR_INPUT
    Enable	: BOOL;
    Enable_Positive	: BOOL;
    Enable_Negative	: BOOL;
    Override	: LREAL ;
    BufferMode	: MC_BufferMode;
END_VAR
END_METHOD

PROPERTY PowerActive : BOOL
GET
END_GET
END_PROPERTY

METHOD PowerEnables
VAR_INPUT
    Enable	: BOOL;
    Enable_Positive	: BOOL;
    Enable_Negative	: BOOL;
END_VAR
END_METHOD

PROPERTY PowerIsEnabled : BOOL
GET
END_GET
END_PROPERTY

PROPERTY PowerOverride : LREAL
GET
END_GET
END_PROPERTY

METHOD ReadAxisParams
VAR_INPUT
    Enable: BOOL;
    RefreshDelay: TIME;
END_VAR
END_METHOD

METHOD Reset
VAR_INPUT
	Execute : BOOL;
END_VAR
END_METHOD

PROPERTY ResetBusy : BOOL
GET
END_GET
END_PROPERTY

PROPERTY ResetDone : BOOL
GET
END_GET
END_PROPERTY

PROPERTY RestoreDone : BOOL
GET
END_GET
END_PROPERTY

METHOD SaveAxisParams
VAR_INPUT
    Enable	: BOOL;
END_VAR
END_METHOD

PROPERTY SavedPosition : LREAL
GET
END_GET
END_PROPERTY

PROPERTY ScaledEncoderCount : UDINT
GET
END_GET
END_PROPERTY

{warning 'Add property implementation'}
PROPERTY StandStill : BOOL
GET
END_GET
END_PROPERTY

(*
    Check all post condition before updating bCommandedMoveAbsolute
    The implmentatation will depend on the axis type
    DS402 NC/Direct axis : Implementation need to check that the drive is in the correct mode before initaiting the move then set bCommandedMoveAbsolute
    MP NC axis : will immediately write to bCommandedMoveAbsolute
*)
METHOD StartMove
VAR_INPUT
    MoveMode	: E_EpicsMotorCmd;
    CmdExecute	: BOOL;
END_VAR
END_METHOD

PROPERTY Stopped : BOOL
GET
END_GET
END_PROPERTY

END_INTERFACE

// ---- POUs/ITFs/I_MotionAxisDS402.TcIO
INTERFACE I_MotionAxisDS402 EXTENDS I_MotionAxis

METHOD ModeOfOperation : BOOL;
VAR_INPUT
    RecentModeOfOperation : E_DS402OpMode;
END_VAR
END_METHOD

END_INTERFACE

// ---- POUs/ITFs/I_MotionDrive.TcIO
INTERFACE I_MotionDrive

METHOD ClearVars
VAR_INPUT
    Done : BOOL;
END_VAR
END_METHOD

PROPERTY EnableMode : ENUM_StageEnableMode
GET
END_GET
SET
END_SET
END_PROPERTY

PROPERTY Name : STRING
GET
END_GET
SET
END_SET
END_PROPERTY

METHOD PreMoveHandling
VAR_INPUT
END_VAR
END_METHOD

METHOD RestoreSettings
VAR_INPUT
END_VAR
END_METHOD

METHOD  UpdateParamAndStatus
VAR_INPUT
END_VAR
END_METHOD

END_INTERFACE

// ---- POUs/ITFs/I_MotionInterlocks.TcIO
// User API for interlocks, add each new interlocks interface here
INTERFACE I_MotionInterlocks

METHOD AxisStatus
VAR_INPUT
	HomeBusy: BOOL;
	PositiveDirection : BOOL;
	NegativeDirection : BOOL;
END_VAR
END_METHOD

METHOD DriveCommands
VAR_INPUT
    MoveEnable: BOOL;
    NewMoveReq : BOOL;
END_VAR
END_METHOD

PROPERTY Error : BOOL
GET
END_GET
END_PROPERTY

PROPERTY ErrorID : UDINT
GET
END_GET
END_PROPERTY

PROPERTY HomeSensor : BOOL
GET
END_GET
END_PROPERTY

PROPERTY Message : T_MAXSTRING
GET
END_GET
END_PROPERTY

PROPERTY MoveBackwardEnabled : BOOL
GET
END_GET
END_PROPERTY

PROPERTY MoveForwardEnabled : BOOL
GET
END_GET
END_PROPERTY

PROPERTY MoveOk : BOOL
GET
END_GET
END_PROPERTY

PROPERTY PowerEnabled : BOOL
GET
END_GET
END_PROPERTY

METHOD Reset
VAR_INPUT
END_VAR
END_METHOD

PROPERTY Warning : BOOL
GET
END_GET
END_PROPERTY

END_INTERFACE

// ---- POUs/ITFs/I_MoveAbsolute.TcIO
INTERFACE I_MoveAbsolute

PROPERTY CommandMoveAbsolute : BOOL
SET
END_SET
END_PROPERTY

METHOD MoveAbsolute
VAR_INPUT
    Execute     : BOOL;
    Position	: LREAL;
    Velocity	: LREAL;
    Acceleration	: LREAL := 0.0;
    Deceleration	: LREAL := 0.0;
    Jerk	: LREAL := 0.0;
    BufferMode	: MC_BufferMode := MC_BufferMode.MC_Aborting;
END_VAR
END_METHOD

PROPERTY MoveAbsoluteAborted : BOOL
GET
END_GET
END_PROPERTY

PROPERTY MoveAbsoluteActive : BOOL
GET
END_GET
END_PROPERTY

PROPERTY MoveAbsoluteBusy : BOOL
GET
END_GET
END_PROPERTY

PROPERTY MoveAbsoluteDone : BOOL
GET
END_GET
END_PROPERTY

PROPERTY MoveAbsoluteError : BOOL
GET
END_GET
END_PROPERTY

PROPERTY MoveAbsoluteErrorID : UDINT
GET
END_GET
END_PROPERTY

END_INTERFACE

// ---- POUs/ITFs/I_Power.TcIO
INTERFACE I_Power  EXTENDS I_Output

METHOD Enables
VAR_INPUT
    Enable	: BOOL;
    Enable_Positive	: BOOL;
    Enable_Negative	: BOOL;
END_VAR
END_METHOD

PROPERTY IsEnabled : BOOL
GET
END_GET
END_PROPERTY

METHOD Power
VAR_INPUT
    Enable	: BOOL;
    Enable_Positive	: BOOL;
    Enable_Negative	: BOOL;
    Override	: LREAL := 100.0;
    BufferMode	: MC_BufferMode := MC_BufferMode.MC_Aborting;
END_VAR
END_METHOD

END_INTERFACE

// ---- POUs/ITFs/I_ReadParameter.TcIO
INTERFACE I_ReadParameter EXTENDS I_Output

PROPERTY AxisReadParamsInit : BOOL
GET
END_GET
END_PROPERTY

METHOD ReadParameters
VAR_INPUT
    Enable: BOOL;
    RefreshDelay: TIME;
END_VAR
END_METHOD

PROPERTY RefVeloSearch : LREAL
GET
END_GET
END_PROPERTY

PROPERTY RefVeloSync : LREAL
GET
END_GET
END_PROPERTY

END_INTERFACE

// ---- POUs/ITFs/I_Reset.TcIO
INTERFACE I_Reset

METHOD Reset
VAR_INPUT
	Execute : BOOL;
END_VAR
END_METHOD

PROPERTY ResetBusy : BOOL
GET
END_GET
END_PROPERTY

PROPERTY ResetDone : BOOL
GET
END_GET
END_PROPERTY

PROPERTY ResetError : BOOL
GET
END_GET
END_PROPERTY

PROPERTY ResetErrorID : UDINT
GET
END_GET
END_PROPERTY

END_INTERFACE

// ---- Test/PRG_TEST.TcPOU
PROGRAM PRG_TEST
VAR
    // New Motion Architecture tests
    fb_BrakeNC_Test: FB_BrakeNC_Test;
 	fb_MoveRequest_Test : FB_MoveRequest_Test;
	fb_MotionInterlocksCommon_Test : FB_MotionInterlocksCommon_Test;
	fb_MotionInterlocksLimSw_Test : FB_MotionInterlocksLimSw_Test;
	fb_MotionLogger_Test : FB_MotionLogger_Test;
	fb_MotionDriveStateMachine_Test : FB_MotionDriveStateMachine_Test;
	fb_MotionDrive_Test : FB_MotionDrive_Test;
// 
    {attribute 'TcNcAxis' := '
        .fbAxisRef[1] := Axes_MotionAxis_Test1;
        .fbAxisRef[2] := Axes_MotionAxis_Test2;
        .fbAxisRef[3] := Axes_MotionAxis_Test3;
        .fbAxisRef[4] := Axes_MotionAxis_Test4;
        .fbAxisRef[5] := Axes_MotionAxis_Test5;
        .fbAxisRef[6] := Axes_MotionAxis_Test6;
        .fbAxisRef[7] := Axes_MotionAxis_Test7;
        .fbAxisRef[8] := Axes_MotionAxis_Test8;
        .fbAxisRef[9] := Axes_MotionAxis_Test9;
        .fbAxisRef[10] := Axes_MotionAxis_Test10;
        .fbAxisRef[11] := Axes_MotionAxis_Test11;
        .fbAxisRef[12] := Axes_MotionAxis_Test12;
        .fbAxisRef[13] := Axes_MotionAxis_Test13;
        .fbAxisRef[14] := Axes_MotionAxis_Test14;
        .fbAxisRef[15] := Axes_MotionAxis_Test15;
        .fbAxisRef[16] := Axes_MotionAxis_Test16
    '}	
	fb_NcMotionBlocks_Test:  FB_NcMotionBlocks_Test;
    {attribute 'TcNcAxis' := '
        .fbAxisRef := Axes_MotionAxis_Test17
    '}	
   	fb_MotionAxisNC_Test : FB_MotionAxisNC_Test;
// 	
    {attribute 'TcNcAxis' := '
        .fbAxisRef[1] := Axis_MotionStageNC_Test1;
        .fbAxisRef[2] := Axis_MotionStageNC_Test2;
        .fbAxisRef[3] := Axis_MotionStageNC_Test3;
        .fbAxisRef[4] := Axis_MotionStageNC_Test4;
        .fbAxisRef[5] := Axis_MotionStageNC_Test5;
        .fbAxisRef[6] := Axis_MotionStageNC_Test6;
        .fbAxisRef[7] := Axis_MotionStageNC_Test7;
        .fbAxisRef[8] := Axis_MotionStageNC_Test8;
	    .fbAxisRef[9] := Axis_MotionStageNC_Test9;
	    .fbAxisRef[10] := Axis_MotionStageNC_Test10;
	    .fbAxisRef[11] := Axis_MotionStageNC_Test11;
	    .fbAxisRef[12] := Axis_MotionStageNC_Test12;
	    .fbAxisRef[13] := Axis_MotionStageNC_Test13;
	    .fbAxisRef[14] := Axis_MotionStageNC_Test14;
	    .fbAxisRef[15] := Axis_MotionStageNC_Test15;
	    .fbAxisRef[16] := Axis_MotionStageNC_Test16;
	    .fbAxisRef[17] := Axis_MotionStageNC_Test17
    '}
 	fb_MotionStageNC_Test :  FB_MotionStageNC_Test;

END_VAR

TcUnit.Run();

END_PROGRAM

// ---- Test/Orchetration/FB_MoveRequest_Test.TcPOU
FUNCTION_BLOCK FB_MoveRequest_Test EXTENDS FB_TestSuite
VAR
        stMotionCommand :  ARRAY[1..10] OF ST_MotionCommand;
		stMotionStatus :  ARRAY[1..10] OF ST_MotionStatus;
END_VAR

GivenMoveRequestAndInterlockAndErrorStatusUpdateRequestStatus_Test1();
GivenMoveRequestDisabledWhenInterlockFalseAlwaysMode_Test2();
GivenAlwaysModeEnableWhenInterlockTrue_Test3();
GivenDuringMotionDisableWhenInterlockFalse_Test4();
GivenDuringMotionEnableWhenInterlockTrue_Test5();
GivenAbsoluteMoveCorrectFlags_Test6();
GivenHomeMoveCorrectFlags_Test7();
GivenInitMoveRequestSetsBusyClearsDoneAndErrorMsg_Test8();
GivenExecuteFlagsSetAndCleared_Test9();

METHOD PRIVATE GivenAbsoluteMoveCorrectFlags_Test6
VAR_INST
    fbMoveRequest : FB_EpicsMoveRequest(
		stMotionCommand:=stMotionCommand[7],
		stMotionStatus:=stMotionStatus[7]
	);
	eExpectedMoveMode :E_EpicsMotorCmd := E_EpicsMotorCmd.MOVE_ABSOLUTE;
END_VAR
// ----------- Absolute Move Command: flags and mode correctness -------------
TEST(__POUNAME());

fbMoveRequest.MoveRequestCmds(
    HomeCmd    := FALSE,
    MoveCmd    := TRUE,
    MoveOk     := TRUE,
    EnableDone := TRUE,
    HomeMode   := E_EpicsHomeCmd.NONE,
    EnableMode := E_StageEnableMode.DURING_MOTION
);
fbMoveRequest();

AssertTrue(fbMoveRequest.Status.bNewMoveReq, 'Should register move request');
AssertTrue(fbMoveRequest.Status.bExecMove, 'Should be ready for move');
AssertFalse(fbMoveRequest.Status.bExecHome, 'Should not be ready for home');
AssertEquals_INT(eExpectedMoveMode, fbMoveRequest.Status.nCommand, 'Command=absolute');
TEST_FINISHED();
END_METHOD

METHOD PRIVATE GivenAlwaysModeEnableWhenInterlockTrue_Test3
VAR_INST
    fbMoveRequest : FB_EpicsMoveRequest(
		stMotionCommand:=stMotionCommand[4],
		stMotionStatus:=stMotionStatus[4]
	);
END_VAR
// ----------- Always mode: should enable if interlock met -------------
TEST(__POUNAME());

fbMoveRequest.MoveRequestCmds(
    HomeCmd    := FALSE,
    MoveCmd    := TRUE,
    MoveOk     := TRUE,
    EnableDone := TRUE,
    HomeMode   := E_EpicsHomeCmd.NONE,
    EnableMode := E_StageEnableMode.ALWAYS
);
fbMoveRequest();

AssertTrue( fbMoveRequest.Status.bEnable, 'Should be enabled when MoveOk is TRUE in ALWAYS mode' );
TEST_FINISHED();
END_METHOD

METHOD PRIVATE GivenDuringMotionDisableWhenInterlockFalse_Test4
VAR_INST
    fbMoveRequest : FB_EpicsMoveRequest(
		stMotionCommand:=stMotionCommand[5],
		stMotionStatus:=stMotionStatus[5]
	);
END_VAR
// ----------- DuringMotion: Must not enable if interlock not met -------------
TEST(__POUNAME());
fbMoveRequest.MoveRequestCmds(
    HomeCmd    := FALSE,
    MoveCmd    := TRUE,
    MoveOk     := FALSE,
    EnableDone := TRUE,
    HomeMode   := E_EpicsHomeCmd.NONE,
    EnableMode := E_StageEnableMode.DURING_MOTION
);
fbMoveRequest();

AssertFalse(fbMoveRequest.Status.bEnable, 'Request disabled if MoveOk is FALSE in DURING_MOTION mode');
TEST_FINISHED();
END_METHOD

METHOD PRIVATE GivenDuringMotionEnableWhenInterlockTrue_Test5
VAR_INST
    fbMoveRequest : FB_EpicsMoveRequest(
		stMotionCommand:=stMotionCommand[6],
		stMotionStatus:=stMotionStatus[6]
	);
END_VAR
TEST(__POUNAME());

fbMoveRequest.MoveRequestCmds(
    HomeCmd    := FALSE,
    MoveCmd    := TRUE,
    MoveOk     := TRUE,
    EnableDone := TRUE,
    HomeMode   := E_EpicsHomeCmd.NONE,
    EnableMode := E_StageEnableMode.DURING_MOTION
);
fbMoveRequest();

AssertTrue(fbMoveRequest.Status.bEnable, 'Request enabled when MoveOk TRUE in DURING_MOTION mode');
TEST_FINISHED();
END_METHOD

METHOD PRIVATE GivenExecuteFlagsSetAndCleared_Test9
VAR_INST
    fbMoveRequest : FB_EpicsMoveRequest(
		stMotionCommand:=stMotionCommand[10],
		stMotionStatus:=stMotionStatus[10]
	);
END_VAR
// ----------- Execute flags set and cleared as expected -------------
TEST(__POUNAME());

	fbMoveRequest.MoveRequestCmds(
		HomeCmd    := FALSE,
		MoveCmd    := TRUE,
		MoveOk     := TRUE,
		EnableDone := TRUE,
		HomeMode   := E_EpicsHomeCmd.NONE,
		EnableMode := E_StageEnableMode.DURING_MOTION
	);
	fbMoveRequest();
	
	AssertTrue(THIS^.stMotionCommand[10].bExecute, 'bExecute must be set');
	AssertTrue(fbMoveRequest.Status.bExecute, 'Local execute flag must be set');
	
	// Simulate user reset/stop
	THIS^.stMotionCommand[10].bExecute := FALSE;
	fbMoveRequest();
	AssertTrue(fbMoveRequest.Status.bPrepareDisable, 'Request must prepare disable after clear');

TEST_FINISHED();
END_METHOD

METHOD PRIVATE GivenHomeMoveCorrectFlags_Test7
VAR_INST
    fbMoveRequest : FB_EpicsMoveRequest(
		stMotionCommand:=stMotionCommand[8],
		stMotionStatus:=stMotionStatus[8]
	);
	nActualMoveMode : INT;
	eExpectedMoveMode :E_EpicsMotorCmd := E_EpicsMotorCmd.HOME;
END_VAR
// ----------- Home Move Command: flags and mode correctness -------------
TEST(__POUNAME());

	fbMoveRequest.MoveRequestCmds(
		HomeCmd    := TRUE,
		MoveCmd    := FALSE,
		MoveOk     := TRUE,
		EnableDone := TRUE,
		HomeMode   := E_EpicsHomeCmd.LOW_LIMIT,
		EnableMode := E_StageEnableMode.DURING_MOTION
	);
	fbMoveRequest();
	
	nActualMoveMode := fbMoveRequest.Status.nCommand;
	AssertTrue(fbMoveRequest.Status.bNewMoveReq, 'Registered home request');
	AssertFalse(fbMoveRequest.Status.bExecMove, 'Should not be absolute for home');
	AssertTrue(fbMoveRequest.Status.bExecHome, 'Home move must be ready');
	AssertEquals_INT(eExpectedMoveMode, nActualMoveMode, 'Command=home');
TEST_FINISHED();
END_METHOD

METHOD PRIVATE GivenInitMoveRequestSetsBusyClearsDoneAndErrorMsg_Test8
VAR_INST
    fbMoveRequest : FB_EpicsMoveRequest(
		stMotionCommand:=stMotionCommand[9],
		stMotionStatus:=stMotionStatus[9]
	);
	sMoveMessage : STRING := '';
END_VAR
// ----------- Init should set busy, clear done, clear error string -------------
TEST(__POUNAME());

	fbMoveRequest.MoveRequestCmds(
		HomeCmd    := FALSE,
		MoveCmd    := TRUE,
		MoveOk     := TRUE,
		EnableDone := TRUE,
		HomeMode   := E_EpicsHomeCmd.NONE,
		EnableMode := E_StageEnableMode.DURING_MOTION
	);

	fbMoveRequest.InitMoveRequest();
	fbMoveRequest();
	
	AssertTrue(stMotionStatus[9].bBusy, 'Busy at init');
	AssertFalse(stMotionStatus[9].bDone, 'Done reset at init');
	AssertEquals_STRING(sMoveMessage, stMotionStatus[9].sErrorMessage, 'Error cleared at init');
TEST_FINISHED();
END_METHOD

METHOD PRIVATE GivenMoveRequestAndInterlockAndErrorStatusUpdateRequestStatus_Test1
VAR_INST
    fbMoveRequest : FB_EpicsMoveRequest(stMotionCommand:=stMotionCommand[1], stMotionStatus:=stMotionStatus[1]);
    eExpectedMoveMode : INT := E_EpicsMotorCmd.MOVE_ABSOLUTE;
    eActualMoveMode : INT;
    sMoveMessage : STRING := '';
END_VAR
TEST(__POUNAME());

	// ------------------------
	// ALWAYS mode: request should only enable when allowed, and latch off on error
	// ------------------------
	fbMoveRequest.MoveRequestCmds(
		HomeCmd := FALSE,
		MoveCmd := FALSE,
		MoveOk := FALSE,
		EnableDone := FALSE,
		HomeMode := E_EpicsHomeCmd.NONE,
		EnableMode := E_StageEnableMode.ALWAYS
	);
	fbMoveRequest();
	
	AssertFalse(
		fbMoveRequest.Status.bEnable,
		'move request must be disabled with invalid interlock in ALWAYS mode #1'
	);
	
	fbMoveRequest.MoveRequestCmds(
		HomeCmd := FALSE,
		MoveCmd := TRUE,
		MoveOk := TRUE,
		EnableDone := TRUE,
		HomeMode := E_EpicsHomeCmd.NONE,
		EnableMode := E_StageEnableMode.ALWAYS
	);
	fbMoveRequest();
	
	AssertTrue(
		fbMoveRequest.Status.bEnable,
		'move request must be enabled with valid interlock in ALWAYS mode #2'
	);
	
	// Now simulate a persistent/latching error after enable
	fbMoveRequest.ClearMoveRequest();
	fbMoveRequest();
	
	stMotionstatus[1].bError := TRUE; // Simulate latching error
	fbMoveRequest.MoveRequestCmds(
		HomeCmd := FALSE,
		MoveCmd := TRUE,
		MoveOk := TRUE,
		EnableDone := TRUE,
		HomeMode := E_EpicsHomeCmd.NONE,
		EnableMode := E_StageEnableMode.ALWAYS
	);
	fbMoveRequest();
	
	AssertFalse(
		fbMoveRequest.Status.bEnable,
		'Latching error condition must disable move request in ALWAYS mode #3'
	);
	
	// ------------------------
	// DURING_MOTION mode: only enable when MoveOk, must stay off with error or missing enables
	// ------------------------
	// 
	// Clear previous request
	fbMoveRequest.ClearMoveRequest();
	fbMoveRequest.ClearMoveRequestErrors();
	fbMoveRequest();
	
	fbMoveRequest.MoveRequestCmds(
		HomeCmd := FALSE,
		MoveCmd := TRUE,
		MoveOk := FALSE,
		EnableDone := FALSE,
		HomeMode := E_EpicsHomeCmd.NONE,
		EnableMode := E_StageEnableMode.DURING_MOTION
	);
	fbMoveRequest();
	
	AssertFalse(
		fbMoveRequest.Status.bEnable,
		'Missing MoveOk must keep move disabled in DURING_MOTION mode #4'
	);
	
	fbMoveRequest.ClearMoveRequest();
	fbMoveRequest();
	
	fbMoveRequest.MoveRequestCmds(
		HomeCmd := FALSE,
		MoveCmd := TRUE,
		MoveOk := TRUE,
		EnableDone := FALSE,
		HomeMode := E_EpicsHomeCmd.NONE,
		EnableMode := E_StageEnableMode.DURING_MOTION
	);
	fbMoveRequest();
	
	AssertTrue(
		fbMoveRequest.Status.bEnable,
		'Move request must be enabled in DURING_MOTION mode #6'
	);
	
	fbMoveRequest.ClearMoveRequest();
	fbMoveRequest();
	
	fbMoveRequest.MoveRequestCmds(
		HomeCmd := FALSE,
		MoveCmd := TRUE,
		MoveOk := TRUE,
		EnableDone := TRUE,
		HomeMode := E_EpicsHomeCmd.NONE,
		EnableMode := E_StageEnableMode.DURING_MOTION
	);
	fbMoveRequest();
	
	eExpectedMoveMode := E_EpicsMotorCmd.MOVE_ABSOLUTE;
	
	AssertTrue(fbMoveRequest.Status.bNewMoveReq, 'Move request must be Registered #7');
	AssertTrue(fbMoveRequest.Status.bExecMove, 'Absolute move must be ready #8');
	AssertFalse(fbMoveRequest.Status.bExecHome, 'Move is not a Homing move #9');
	AssertEquals_INT(eExpectedMoveMode, fbMoveRequest.Status.nCommand, 'Move command must be absolute #10');
	
	fbMoveRequest.ClearMoveRequest();
	fbMoveRequest();
	
	fbMoveRequest.MoveRequestCmds(
		HomeCmd := TRUE,
		MoveCmd := FALSE,
		MoveOk := TRUE,
		EnableDone := TRUE,
		HomeMode := E_EpicsHomeCmd.LOW_LIMIT,
		EnableMode := E_StageEnableMode.DURING_MOTION
	);
	fbMoveRequest();
	
	eExpectedMoveMode := E_EpicsMotorCmd.HOME;
	eActualMoveMode := fbMoveRequest.Status.nCommand;
	
	AssertTrue(fbMoveRequest.Status.bNewMoveReq, 'Move request must be Registered #11');
	AssertFalse(fbMoveRequest.Status.bExecMove, 'Move is not Absolute #12');
	AssertTrue(fbMoveRequest.Status.bExecHome, 'Home move must be ready #13');
	AssertEquals_INT(eExpectedMoveMode, eActualMoveMode, 'Move command must be a valid homing mode #14');
	
	fbMoveRequest.ClearMoveRequest();
	fbMoveRequest();
	
	stMotionstatus[1].bError := FALSE;
	fbMoveRequest.MoveRequestCmds(
		HomeCmd := FALSE,
		MoveCmd := TRUE,
		MoveOk := TRUE,
		EnableDone := TRUE,
		HomeMode := E_EpicsHomeCmd.NONE,
		EnableMode := E_StageEnableMode.DURING_MOTION
	);
	fbMoveRequest.InitMoveRequest();
	fbMoveRequest();
	
	AssertTrue(stMotionstatus[1].bBusy, 'Move Request Busy flag must be set at init #15');
	AssertFalse(stMotionstatus[1].bDone, 'Move request Done flag must reset at init #16');
	AssertEquals_STRING(sMoveMessage, stMotionstatus[1].sErrorMessage, 'Move request Error flag must be cleared at init #17');
	
	fbMoveRequest.ClearMoveRequest();
	fbMoveRequest();
	
	stMotionstatus[1].bError := FALSE;
	fbMoveRequest.MoveRequestCmds(
		HomeCmd := FALSE,
		MoveCmd := TRUE,
		MoveOk := TRUE,
		EnableDone := TRUE,
		HomeMode := E_EpicsHomeCmd.NONE,
		EnableMode := E_StageEnableMode.DURING_MOTION
	);
	fbMoveRequest();
	
	AssertTrue(THIS^.stMotionCommand[1].bExecute, 'Execute must be set by now #18');
	AssertTrue(fbMoveRequest.Status.bExecute, 'Local Execute must be set by now #19');
	
	// Simulate user stop
	THIS^.stMotionCommand[1].bExecute := FALSE;
	fbMoveRequest();
	
	AssertTrue(fbMoveRequest.Status.bPrepareDisable, 'Must be preparing to disable by now #20');

TEST_FINISHED();
END_METHOD

METHOD PRIVATE GivenMoveRequestDisabledWhenInterlockFalseAlwaysMode_Test2
VAR_INST
    fbMoveRequest : FB_EpicsMoveRequest(
		stMotionCommand:=stMotionCommand[3],
		stMotionStatus:=stMotionStatus[3]
	);
END_VAR
// ----------- Always mode: should NOT enable if interlock not met -------------
TEST(__POUNAME());
	
	fbMoveRequest.MoveRequestCmds(
		HomeCmd    := FALSE,
		MoveCmd    := FALSE,
		MoveOk     := FALSE,
		EnableDone := FALSE,
		HomeMode   := E_EpicsHomeCmd.NONE,
		EnableMode := E_StageEnableMode.ALWAYS
	);
	fbMoveRequest();
	
	AssertFalse(fbMoveRequest.Status.bEnable, 'Should be disabled if MoveOk is FALSE in ALWAYS mode');
TEST_FINISHED();
END_METHOD

END_FUNCTION_BLOCK

// ---- Test/Interlok/FB_MotionInterlocksCommon_Test.TcPOU
FUNCTION_BLOCK FB_MotionInterlocksCommon_Test EXTENDS FB_TestSuite
VAR
    fbMotionLogger 		: ARRAY[1..5] OF FB_MotionLogger;
END_VAR

GivenEpicsEnableAndHardwareEnableIfNotUserEnableThenResetPowerEnableAndMoveOk_Test1();
GivenEpicsEnablehardwareEnableAndUserEnableUpdatePowerEnableAndMoveOk_Test2();
GivenhardwareEnableAndUserEnableIfNotEpicsEnableResetPowerEnable_Test3();
GivenUserEnableAndNothardwareEnableThenSetHardwareEnableErrorResetMoveOk_Test4();
GivenInterlockEventIFGlobalResetClearErrors_Test5();

METHOD PRIVATE GivenEpicsEnableAndHardwareEnableIfNotUserEnableThenResetPowerEnableAndMoveOk_Test1
VAR
    fbMotionInterlocksCommon : FB_MotionInterlocksCommon(
		iMotionLogger:=fbMotionLogger[1]
	);
    sExpectedUserEnableMessage : STRING := 'User enable interlock triggered!';
    sActUserEnableMessage : STRING;
END_VAR
TEST(__POUNAME());
// Test UserEnable interlock trigger
fbMotionInterlocksCommon.EnableInterlocks(UserEnable:=FALSE, HardwareEnable:=TRUE);
fbMotionInterlocksCommon.DriveCommands(MoveEnable:=TRUE, NewMoveReq:=FALSE);
fbMotionInterlocksCommon();

AssertFalse(Condition := fbMotionInterlocksCommon.PowerEnabled,
           Message := 'UserEnbale Interlock triggered PowerEnable must be unset #1');

AssertFalse(Condition := fbMotionInterlocksCommon.MoveOk,
           Message := 'UserEnbale Interlock triggered MoveOk must be unset #2');

sActUserEnableMessage := fbMotionInterlocksCommon.Message;
AssertEquals ( Expected:=sExpectedUserEnableMessage, Actual:=sActUserEnableMessage,
            Message:='Incorrect UserEnbale trigger Error Msg #3');

TEST_FINISHED();
END_METHOD

METHOD PRIVATE GivenEpicsEnablehardwareEnableAndUserEnableUpdatePowerEnableAndMoveOk_Test2
VAR
    fbMotionInterlocksCommon : FB_MotionInterlocksCommon(
		iMotionLogger:=fbMotionLogger[2]
	);
    sExpectedMessage : STRING := '';
    sActMessage : STRING;
    nExpectedErrorId : UDINT := 0;
    nActErrorId : UDINT;
END_VAR
TEST(__POUNAME());
// PowerEnable and MoveOk Set
fbMotionInterlocksCommon.EnableInterlocks(UserEnable:=TRUE, HardwareEnable:=TRUE);
fbMotionInterlocksCommon.DriveCommands(MoveEnable:=TRUE, NewMoveReq:=FALSE);
fbMotionInterlocksCommon();

AssertTrue(Condition := fbMotionInterlocksCommon.PowerEnabled,
           Message := 'Hardware or UserEnable Interlock not set #1');

AssertTrue(Condition := fbMotionInterlocksCommon.MoveOk,
           Message := 'Hardware or UserEnable Interlock not set #2');

AssertFalse(Condition := fbMotionInterlocksCommon.Error,
           Message := 'No Error expected #3');

nActErrorId := fbMotionInterlocksCommon.ErrorID;
AssertEquals ( Expected:=nExpectedErrorId, Actual:=nActErrorId ,
            Message:='ErrorID must be 0 #4');

sActMessage := fbMotionInterlocksCommon.Message;
AssertEquals ( Expected:=sExpectedMessage, Actual:=sActMessage ,
            Message:='No error Message #5');

TEST_FINISHED();
END_METHOD

METHOD PRIVATE GivenhardwareEnableAndUserEnableIfNotEpicsEnableResetPowerEnable_Test3
VAR
    fbMotionInterlocksCommon : FB_MotionInterlocksCommon(
		iMotionLogger:=fbMotionLogger[3]
	);
    sExpectedMessage : STRING := '';
    sActMessage : STRING;
    nExpectedErrorId : UDINT := 0;
    nActErrorId : UDINT;
END_VAR
TEST(__POUNAME());

fbMotionInterlocksCommon.EnableInterlocks(UserEnable:=TRUE, HardwareEnable:=TRUE);
fbMotionInterlocksCommon.DriveCommands(MoveEnable:=FALSE, NewMoveReq:=FALSE);
fbMotionInterlocksCommon();

AssertFalse(Condition := fbMotionInterlocksCommon.PowerEnabled,
           Message := 'No Epics Enable, PowerEnabled must not be set #1');

AssertTrue(Condition := fbMotionInterlocksCommon.MoveOk,
           Message := 'Epics Enable reset, Move Request must be invalid #2');

AssertFalse(Condition := fbMotionInterlocksCommon.Error,
           Message := 'No Error expected #3');

nActErrorId := fbMotionInterlocksCommon.ErrorID;
AssertEquals ( Expected:=nExpectedErrorId, Actual:=nActErrorId ,
            Message:='ErrorID must be 0 #4');

sActMessage := fbMotionInterlocksCommon.Message;
AssertEquals ( Expected:=sExpectedMessage, Actual:=sActMessage ,
            Message:='No error Message #5');
TEST_FINISHED();
END_METHOD

METHOD PRIVATE GivenInterlockEventIFGlobalResetClearErrors_Test5
VAR
     fbMotionInterlocksCommon : FB_MotionInterlocksCommon(
		iMotionLogger:=fbMotionLogger[5]
	);
    sExpectedMessage : STRING := '';
    sActMessage : STRING;
    nExpectedErrorId : UDINT := 0;
    nActErrorId : UDINT;
END_VAR
TEST(__POUNAME());
// HardwareEnable unset
fbMotionInterlocksCommon.EnableInterlocks(UserEnable:=TRUE, HardwareEnable:=FALSE);
fbMotionInterlocksCommon.DriveCommands(MoveEnable:=FALSE, NewMoveReq:=FALSE);
fbMotionInterlocksCommon();

AssertTRUE(Condition := fbMotionInterlocksCommon.Error,
           Message := 'HardwareEnable Error must be set #1');

// Test Global Reset to clear internal flags
fbMotionInterlocksCommon.EnableInterlocks(UserEnable:=TRUE, HardwareEnable:=TRUE);
fbMotionInterlocksCommon.Reset();
fbMotionInterlocksCommon();

AssertFalse(Condition := fbMotionInterlocksCommon.Error,
           Message := 'Error must be clear after global reset #2');

sActMessage := fbMotionInterlocksCommon.Message;
AssertEquals ( Expected:=sExpectedMessage, Actual:=sActMessage,
            Message:='Error Msg must be cleared #3');
TEST_FINISHED();
END_METHOD

METHOD PRIVATE GivenUserEnableAndNothardwareEnableThenSetHardwareEnableErrorResetMoveOk_Test4
VAR
    fbMotionInterlocksCommon : FB_MotionInterlocksCommon(
		iMotionLogger:=fbMotionLogger[4]
	);
    sExpectedHardwareEnableMessage : STRING := 'Hardware enable interlock triggered!';
    sActHardwareEnableMessage : STRING;
    nExpectedErrorId : UDINT := 11;
    nActErrorId : UDINT;
END_VAR
TEST(__POUNAME());
// HardwareEnable unset
fbMotionInterlocksCommon.EnableInterlocks(UserEnable:=TRUE, HardwareEnable:=FALSE);
fbMotionInterlocksCommon.DriveCommands(MoveEnable:=TRUE, NewMoveReq:=FALSE);
fbMotionInterlocksCommon();
// 
AssertFalse(Condition := fbMotionInterlocksCommon.PowerEnabled,
           Message := 'Hardware Interlock triggered PowerEnable must be unset #1');

AssertFalse(Condition := fbMotionInterlocksCommon.MoveOk,
           Message := 'Hardware Interlock triggered MoveOk must be unset #2');
// 
AssertTrue(Condition := fbMotionInterlocksCommon.Error,
           Message := 'Hardware Interlock triggered Error must be set #3');

AssertTrue(condition:=nExpectedErrorId = fbMotionInterlocksCommon.ErrorID, Message:='Incorrect Hardware trigger ErrorID #4');

AssertTrue ( condition:=(fbMotionInterlocksCommon.Message = sExpectedHardwareEnableMessage) , Message:='Incorrect Hardware trigger Error Msg #5');

TEST_FINISHED();
END_METHOD

END_FUNCTION_BLOCK

// ---- POUs/FBs/Common/FB_MotionInterlocksCommon.TcPOU
FUNCTION_BLOCK FB_MotionInterlocksCommon IMPLEMENTS I_MotionInterlocksCommon
VAR
    {attribute 'hide'}
    iMotionLogger 		: I_MotionLogger;
    {attribute 'hide'}
    bPowerEnabled: BOOL:=FALSE;
    {attribute 'hide'}
    bMoveEnable: BOOL;
    {attribute 'hide'}
    bReset : BOOL;
    {attribute 'hide'}
    sMessage : STRING;
    {attribute 'hide'}
    bError : BOOL;
    {attribute 'hide'}
    nErrorID : UDINT;
    {attribute 'hide'}
    bMoveOk : BOOL;
    // Used by the IOC to disable an axis
    {attribute 'pytmc' := '
        pv: PLC:bUserEnable
        io: io
        field: ZNAM DISABLE
        field: ONAM ENABLE
        field: DESC Used to disable power entirely for an axis
    '}
    bUserEnable: BOOL := TRUE;	
   // NC STO Input: TRUE if ok to move
    {attribute 'pytmc' := '
        pv: PLC:bHardwareEnable
        io: i
        field: ZNAM FALSE
        field: ONAM TRUE
        field: DESC TRUE if STO not hit
    '}
    bHardwareEnable AT %I*: BOOL ;
	rtError : R_TRIG;
END_VAR

// ===== Interlock and Error Handling Block =====

// 1. Safety: Check logger
IF (iMotionLogger = 0) THEN
    // Optionally: set error status in status struct for diagnostics!
    RETURN;
END_IF

// 2. Compute power enable
bPowerEnabled := bMoveEnable AND bHardwareEnable AND bUserEnable;

// 3. Compute move OK
bMoveOk := bUserEnable AND bHardwareEnable;

// 4. Interlock error condition
IF NOT bUserEnable OR NOT bHardwareEnable THEN
    bError := TRUE;
    nErrorID := 11;
    bMoveOk := FALSE;

    IF NOT bUserEnable THEN
        sMessage := 'User enable interlock triggered!';
    ELSE
        sMessage := 'Hardware enable interlock triggered!';
    END_IF
END_IF

// 5. Log error on edge (only when error flips TRUE)
rtError(CLK := bError);
IF rtError.Q THEN
    iMotionLogger.Logger(
        Message := sMessage,
        Level := E_MotionLogLevel.ERROR,
        Source := 'MotionInterlocksCommon'
    );    
END_IF

METHOD PUBLIC CallAfterInit
VAR_INPUT	
    iMotionLogger : I_MotionLogger;
END_VAR
THIS^.iMotionLogger := iMotionLogger;
END_METHOD

METHOD DriveCommands
VAR_INPUT
    MoveEnable: BOOL;
    NewMoveReq : BOOL;
END_VAR
THIS^.bMoveEnable:=MoveEnable;
END_METHOD

METHOD EnableInterlocks
VAR_INPUT
	UserEnable : BOOL;
	HardwareEnable : BOOL;
END_VAR
bUserEnable := UserEnable;
bHardwareEnable := HardwareEnable;
END_METHOD

{attribute 'monitoring' := 'variable'}
PROPERTY Error : BOOL
GET
Error := bError;
END_GET
END_PROPERTY

PROPERTY ErrorID : UDINT
GET
ErrorID := nErrorID;
END_GET
END_PROPERTY

//FB_Init is always available implicitly and it is used primarily for initialization.
//The return value is not evaluated. For a specific influence, you can also declare the
//methods explicitly and provide additional code there with the standard initialization
//code. You can evaluate the return value.
METHOD FB_Init: BOOL
VAR_INPUT
    bInitRetains: BOOL; // TRUE: the retain variables are initialized (reset warm / reset cold)
    bInCopyCode: BOOL;  // TRUE: the instance will be copied to the copy code afterward (online change)
    iMotionLogger 		: I_MotionLogger;
END_VAR
THIS^.iMotionLogger := iMotionLogger;
END_METHOD

PROPERTY Message : T_MAXSTRING
GET
Message := sMessage;
END_GET
END_PROPERTY

{attribute 'monitoring' := 'variable'}
PROPERTY MoveOk : BOOL
GET
MoveOk := bMoveOk;
END_GET
END_PROPERTY

{attribute 'monitoring' := 'variable'}
PROPERTY PowerEnabled : BOOL
GET
PowerEnabled :=bPowerEnabled;
END_GET
END_PROPERTY

METHOD Reset
THIS^.bError := FALSE;
THIS^.nErrorID:= 0;
THIS^.sMessage:='';
END_METHOD

END_FUNCTION_BLOCK

// ---- Test/Interlok/FB_MotionInterlocksLimSw_Test.TcPOU
FUNCTION_BLOCK INTERNAL FB_MotionInterlocksLimSw_Test EXTENDS FB_TestSuite
VAR
    fbLimSwStatus: ARRAY [1..6] OF FB_LimSwStatus_testDouble;
    fbMotionInterlocksCommon:  ARRAY [1..6] OF  FB_MotionInterlocksCommon_TestDouble;
    fbMotionLogger : ARRAY [1..16] OF FB_MotionLogger_TestDouble;
END_VAR

GivenPositiveLimHitEventIfGlobalResetOrNewMoveReqClearLocalFlags_Test1();
GivenLimSwStatusEventIfStandStillUpdateBackwardAndFowardEnable_Test2();
GivenCommonInterlockErrorsThenSetLocalErrors_Test3();
GivenLimForwardAndBackwardActiveAxisMovingInNegativeDirectionIfPosiveLimishitThenNoLimHitEvent_Test4();
GivenLimForwardAndBackwardActiveAxisMovingInPosiveDirectionIfPosiveLimishitThenLimHitEventOccured_test5();
GivenLimSwStatusActiveAndAxisHomingInPosOrNegDirectionThenNoLimHitEvent_Test6();

METHOD PRIVATE GivenCommonInterlockErrorsThenSetLocalErrors_Test3
VAR_INST
    nExpectedErrorId: UDINT := 1;
    nActErrorId: UDINT;
    sExpectedMessage: STRING := 'User enable interlock triggered!';
    sActMessage: STRING;
    // subject under test
    fbMotionInterlocksLimSw : FB_MotionInterlocksLimSw(
		iMotionInterlocksCommon:=fbMotionInterlocksCommon[3], 
		iLimSwStatus:=fbLimSwStatus[3],
		iMotionLogger := fbMotionLogger[3]
	);
END_VAR
TEST(__POUNAME());
// Test UserEnable interlock trigger
fbMotionInterlocksCommon[3].Error := TRUE;
fbMotionInterlocksCommon[3].ErrorID:=1;
fbMotionInterlocksCommon[3].Message:=sExpectedMessage;
fbMotionInterlocksCommon[3]();
fbMotionInterlocksLimSw();

AssertTrue(Condition := fbMotionInterlocksLimSw.Error,
           Message := 'Common interlock event must set this error #1');

nActErrorId := fbMotionInterlocksLimSw.ErrorID;
AssertEquals ( Expected:=nExpectedErrorId, Actual:=nActErrorId ,
            Message:='Common interlock event must set this errorId #2');

sActMessage := fbMotionInterlocksLimSw.Message;
AssertEquals ( Expected:=sExpectedMessage, Actual:=sActMessage,
            Message:='Common interlock event must set this error msg #3');

fbMotionInterlocksCommon[3].ResetErrors();
fbMotionInterlocksCommon[3]();
fbMotionInterlocksLimSw();

TEST_FINISHED();
END_METHOD

METHOD PRIVATE GivenLimForwardAndBackwardActiveAxisMovingInNegativeDirectionIfPosiveLimishitThenNoLimHitEvent_Test4
VAR_INST
    tonLimSwStatusEvent : TON := (IN:=TRUE, PT:=T#0S);
    fbMotionInterlocksLimSw : FB_MotionInterlocksLimSw(
		iMotionInterlocksCommon:=fbMotionInterlocksCommon[4], 
		iLimSwStatus:=fbLimSwStatus[4],
		iMotionLogger := fbMotionLogger[4]
	);
END_VAR
TEST(__POUNAME());
tonLimSwStatusEvent();
fbLimSwStatus[4].LimitForwardEnable := TRUE;
fbLimSwStatus[4].LimitBackwardEnable := TRUE;
fbLimSwStatus[4]();
fbMotionInterlocksLimSw.AxisStatus(HomeBusy:=FALSE, PositiveDirection:=FALSE, NegativeDirection:=TRUE);
fbMotionInterlocksLimSw();


IF tonLimSwStatusEvent.Q THEN
    fbLimSwStatus[4].LimitForwardEnable := FALSE;
    fbLimSwStatus[4]();
    tonLimSwStatusEvent.IN:=FALSE;
END_IF

fbMotionInterlocksLimSw();

AssertFalse(Condition := fbMotionInterlocksLimSw.Warning,
           Message := 'No Warning event expected #1');
AssertFalse(Condition := fbMotionInterlocksLimSw.LimHit,
           Message := 'No Lim Hit event expected #2');
TEST_FINISHED();
END_METHOD

METHOD PRIVATE  GivenLimForwardAndBackwardActiveAxisMovingInPosiveDirectionIfPosiveLimishitThenLimHitEventOccured_Test5
VAR_INST
    tonLimSwStatusEvent : TON := (IN:=TRUE, PT:=T#0S);
    fbMotionInterlocksLimSw : FB_MotionInterlocksLimSw(
		iMotionInterlocksCommon:=fbMotionInterlocksCommon[5], 
		iLimSwStatus:=fbLimSwStatus[5],
		iMotionLogger := fbMotionLogger[5]
	);
END_VAR
TEST(__POUNAME());
tonLimSwStatusEvent();
fbLimSwStatus[5].LimitForwardEnable := TRUE;
fbLimSwStatus[5].LimitBackwardEnable := TRUE;
fbMotionInterlocksLimSw.AxisStatus(HomeBusy:=FALSE, PositiveDirection:=TRUE, NegativeDirection:=FALSE);
fbLimSwStatus[5]();
fbMotionInterlocksLimSw();

IF tonLimSwStatusEvent.Q THEN
    fbLimSwStatus[5].LimitForwardEnable := FALSE;
    tonLimSwStatusEvent.IN := FALSE;
END_IF

fbLimSwStatus[5]();
fbMotionInterlocksLimSw();

AssertTrue(Condition := fbMotionInterlocksLimSw.Warning,
                   Message := 'Expecting a Warning event after positive lim hit #1');
AssertTrue(Condition := fbMotionInterlocksLimSw.LimHit,
                   Message := 'Expecting a Limit hit event after positive lim hit #2');
TEST_FINISHED();
END_METHOD

METHOD PRIVATE GivenLimSwStatusActiveAndAxisHomingInPosOrNegDirectionThenNoLimHitEvent_Test6
VAR_INST
    fbMotionInterlocksLimSw : FB_MotionInterlocksLimSw(
		iMotionInterlocksCommon:=fbMotionInterlocksCommon[6], 
		iLimSwStatus:=fbLimSwStatus[6],
		iMotionLogger := fbMotionLogger[6]
	);
END_VAR
TEST(__POUNAME());

fbLimSwStatus[6].LimitForwardEnable := TRUE;
fbLimSwStatus[6].LimitBackwardEnable := TRUE;
fbMotionInterlocksLimSw.AxisStatus(HomeBusy:=TRUE, PositiveDirection:=TRUE, NegativeDirection:=FALSE);
fbLimSwStatus[6]();
fbMotionInterlocksLimSw();

AssertFalse(Condition := fbMotionInterlocksLimSw.Warning,
           Message := 'Warning event while homing unexpected #1');

AssertFalse(Condition := fbMotionInterlocksLimSw.LimHit,
           Message := 'Lim hit event while homing unexpected #2');

fbMotionInterlocksLimSw.AxisStatus(HomeBusy:=TRUE, PositiveDirection:=FALSE, NegativeDirection:=TRUE);
fbLimSwStatus[6]();
fbMotionInterlocksLimSw();

AssertFalse(Condition := fbMotionInterlocksLimSw.Warning,
           Message := 'Warning event while homing unexpected #3');

AssertFalse(Condition := fbMotionInterlocksLimSw.LimHit,
           Message := 'Lim hit event while homing unexpected #4');

TEST_FINISHED();
END_METHOD

METHOD PRIVATE GivenLimSwStatusEventIfStandStillUpdateBackwardAndFowardEnable_Test2
VAR_INST
    fbMotionInterlocksLimSw : FB_MotionInterlocksLimSw(
		iMotionInterlocksCommon:=fbMotionInterlocksCommon[2], 
		iLimSwStatus:=fbLimSwStatus[2],
		iMotionLogger := fbMotionLogger[2]
	);
END_VAR
TEST(__POUNAME());
// Test LimSwStatus Events and update backward and forward Enable
fbLimSwStatus[2].LimitForwardEnable := TRUE;
fbLimSwStatus[2].LimitBackwardEnable := TRUE;
fbMotionInterlocksLimSw.AxisStatus(HomeBusy:=FALSE, PositiveDirection:=FALSE, NegativeDirection:=FALSE);
fbLimSwStatus[2]();
fbMotionInterlocksLimSw();

AssertTrue(Condition := fbMotionInterlocksLimSw.MoveBackwardEnabled,
           Message := 'MoveBackwardEnabled must be set #1');

AssertTrue(Condition := fbMotionInterlocksLimSw.MoveForwardEnabled,
           Message := 'MoveForwardwardEnabled must be set #2');

fbLimSwStatus[2].LimitForwardEnable := FALSE;
fbLimSwStatus[2].LimitBackwardEnable := FALSE;
fbMotionInterlocksLimSw.AxisStatus(HomeBusy:=FALSE, PositiveDirection:=FALSE, NegativeDirection:=FALSE);
fbLimSwStatus[2]();
fbMotionInterlocksLimSw();

AssertFalse(Condition := fbMotionInterlocksLimSw.MoveBackwardEnabled,
           Message := 'MoveBackwardEnabled must not be set #3');

AssertFalse(Condition := fbMotionInterlocksLimSw.MoveForwardEnabled,
           Message := 'MoveForwardwardEnabled must not be set #4');

TEST_FINISHED();
END_METHOD

METHOD PRIVATE GivenPositiveLimHitEventIfGlobalResetOrNewMoveReqClearLocalFlags_Test1
VAR_INST
    fbMotionInterlocksLimSw : FB_MotionInterlocksLimSw(
		iMotionInterlocksCommon:=fbMotionInterlocksCommon[1], 
		iLimSwStatus:=fbLimSwStatus[1],
		iMotionLogger := fbMotionLogger[1]
	);
END_VAR
TEST(__POUNAME());
fbLimSwStatus[1].LimitForwardEnable := TRUE;
fbLimSwStatus[1].LimitBackwardEnable := TRUE;
fbMotionInterlocksLimSw.AxisStatus(HomeBusy:=FALSE, PositiveDirection:=TRUE, NegativeDirection:=FALSE);
fbLimSwStatus[1]();
fbMotionInterlocksLimSw();

// Create Forward limit hit event
fbLimSwStatus[1].LimitForwardEnable := FALSE;
fbLimSwStatus[1]();
fbMotionInterlocksLimSw();

// Reset Flags
fbMotionInterlocksLimSw.Reset();
fbMotionInterlocksLimSw();

AssertFalse(Condition := fbMotionInterlocksLimSw.Warning,
               Message := 'Warning should be cleared #1');
AssertFalse(Condition := fbMotionInterlocksLimSw.LimHit,
               Message := 'Limit hit flag should be cleared #2');




//Rest axis
fbLimSwStatus[1].LimitForwardEnable := TRUE;
fbLimSwStatus[1].LimitBackwardEnable := TRUE;
fbLimSwStatus[1]();
fbMotionInterlocksLimSw.DriveCommands(MoveEnable:=FALSE, NewMoveReq:=FALSE);
fbMotionInterlocksLimSw.AxisStatus(HomeBusy:=FALSE, PositiveDirection:=FALSE, NegativeDirection:=FALSE);
fbMotionInterlocksLimSw();

// Discrete motion in negative direction
fbMotionInterlocksLimSw.AxisStatus(HomeBusy:=FALSE, PositiveDirection:=FALSE, NegativeDirection:=TRUE);
fbMotionInterlocksLimSw();

// Create backward limit hit event
fbLimSwStatus[1].LimitBackwardEnable := FALSE;
fbLimSwStatus[1]();
fbMotionInterlocksLimSw();

// clear Flags from global reset
fbMotionInterlocksLimSw.Reset();
fbMotionInterlocksLimSw();

AssertFalse(Condition := fbMotionInterlocksLimSw.Warning,
               Message := 'Warning should be cleared #3');
AssertFalse(Condition := fbMotionInterlocksLimSw.LimHit,
               Message := 'Limit hit flag should be cleared #4');



//Rest axis
fbLimSwStatus[1].LimitForwardEnable := TRUE;
fbLimSwStatus[1].LimitBackwardEnable := TRUE;
fbLimSwStatus[1]();
fbMotionInterlocksLimSw.DriveCommands(MoveEnable:=FALSE, NewMoveReq:=FALSE);
fbMotionInterlocksLimSw.AxisStatus(HomeBusy:=FALSE, PositiveDirection:=FALSE, NegativeDirection:=FALSE);
fbMotionInterlocksLimSw();

// Discrete motion in positive direction
fbMotionInterlocksLimSw.AxisStatus(HomeBusy:=FALSE, PositiveDirection:=TRUE, NegativeDirection:=FALSE);
fbMotionInterlocksLimSw();

// Create forward limit hit event
fbLimSwStatus[1].LimitForwardEnable := FALSE;
fbLimSwStatus[1]();
fbMotionInterlocksLimSw();

// clear Flags from global reset
fbMotionInterlocksLimSw.DriveCommands(MoveEnable:=FALSE, NewMoveReq:=TRUE);
fbMotionInterlocksLimSw();

AssertFalse(Condition := fbMotionInterlocksLimSw.Warning,
               Message := 'Warning should be cleared #5');
AssertFalse(Condition := fbMotionInterlocksLimSw.LimHit,
               Message := 'Limit hit flag should be cleared #6');

TEST_FINISHED();
END_METHOD

END_FUNCTION_BLOCK

// ---- Test/TestDouble/FB_LimSwStatus_testDouble.TcPOU
FUNCTION_BLOCK FB_LimSwStatus_testDouble IMPLEMENTS I_LimSwStatus
VAR
   // NC Forward Limit Switch: TRUE if ok to move
    bLimitForwardEnable : BOOL := TRUE;
    // NC Backward Limit Switch: TRUE if ok to move
    bLimitBackwardEnable : BOOL := TRUE;
    // NO Home Switch: TRUE if at home
    bHome : BOOL;
END_VAR

PROPERTY LimitBackwardEnable : BOOL
GET
LimitBackwardEnable := bLimitBackwardEnable;
END_GET
SET
bLimitBackwardEnable := LimitBackwardEnable;
END_SET
END_PROPERTY

PROPERTY LimitForwardEnable : BOOL
GET
LimitForwardEnable := bLimitForwardEnable;
END_GET
SET
bLimitForwardEnable := LimitForwardEnable;
END_SET
END_PROPERTY

PROPERTY LimitHome : BOOL
GET
 LimitHome := bHome;
END_GET
SET
 bHome := LimitHome;
END_SET
END_PROPERTY

END_FUNCTION_BLOCK

// ---- Test/TestDouble/FB_MotionInterlocksCommon_TestDouble.TcPOU
FUNCTION_BLOCK FB_MotionInterlocksCommon_TestDouble IMPLEMENTS I_MotionInterlocksCommon
VAR
    bPowerEnabled: BOOL:=FALSE;
   // NC STO Input: TRUE if ok to move
    bHardwareEnable : BOOL ;
    bUserEnable: BOOL := TRUE;
    bEnable: BOOL;
    bReset : BOOL;
    sMessage : STRING;
    bError : BOOL;
    nErrorID : UDINT;
    // Set by default, an error condition will reset this
    bMoveOk : BOOL := TRUE;

END_VAR

METHOD DriveCommands
VAR_INPUT
    MoveEnable: BOOL;
    NewMoveReq : BOOL;
END_VAR
THIS^.bEnable := MoveEnable;
END_METHOD

{warning 'Add method implementation '}
METHOD EnableInterlocks
VAR_INPUT
	UserEnable	: BOOL;
	HardwareEnable	: BOOL;
END_VAR
END_METHOD

PROPERTY Error : BOOL
GET
Error := bError;
END_GET
SET
bError := Error;
END_SET
END_PROPERTY

PROPERTY ErrorID : UDINT
GET
ErrorID := nErrorID;
END_GET
SET
nErrorID := ErrorID;
END_SET
END_PROPERTY

PROPERTY HardwareEnable : BOOL
GET
END_GET
SET
bHardwareEnable := HardwareEnable;
END_SET
END_PROPERTY

PROPERTY Message : T_MAXSTRING
GET
Message := sMessage;
END_GET
SET
sMessage := Message;
END_SET
END_PROPERTY

PROPERTY MoveOk : BOOL
GET
MoveOk := bMoveOk;
END_GET
SET
END_SET
END_PROPERTY

PROPERTY PowerEnabled : BOOL
GET
PowerEnabled :=bPowerEnabled;
END_GET
SET
END_SET
END_PROPERTY

METHOD Reset
END_METHOD

METHOD ResetErrors
VAR_INPUT
END_VAR
bError := FALSE;
nErrorID:= 0;
sMessage:='';
END_METHOD

PROPERTY UserEnable : BOOL
GET
END_GET
SET
bUserEnable := UserEnable;
END_SET
END_PROPERTY

END_FUNCTION_BLOCK

// ---- Test/TestDouble/FB_MotionLogger_TestDouble.TcPOU
FUNCTION_BLOCK FB_MotionLogger_TestDouble IMPLEMENTS I_MotionLogger
VAR
END_VAR

{warning 'Add method implementation '}
METHOD Clear
END_METHOD

METHOD ErrorCodeLookup : STRING
VAR_INPUT
	nErrorId	: UDINT;
END_VAR
END_METHOD

METHOD GetAllMessages :  STRING(1024)
END_METHOD

{warning 'Add method implementation '}
METHOD GetMessageCount : UINT
VAR_OUTPUT
	nCount	: UINT;
END_VAR
END_METHOD

{warning 'Add method implementation '}
METHOD Logger
VAR_INPUT
	Message	: STRING;
	Level	: E_MotionLogLevel := .E_MotionLogLevel.INFO;
	Source	: STRING := '';
END_VAR
END_METHOD

END_FUNCTION_BLOCK

// ---- Test/Utils/FB_MotionLogger_Test.TcPOU
FUNCTION_BLOCK INTERNAL FB_MotionLogger_Test EXTENDS FB_TestSuite

VAR

END_VAR

GetLastWarningMessage_Test1();

METHOD PRIVATE GetLastWarningMessage_Test1
VAR_INST
	logs : STRING(1024);
	fbMotionLogger : FB_MotionLogger(sName:='slitX') ;
END_VAR
TEST(__POUNAME());
fbMotionLogger.Clear();
fbMotionLogger.Logger(Message := 'One', Level := E_MotionLogLevel.INFO, Source := 'A');
fbMotionLogger.Logger(Message := 'Two', Level := E_MotionLogLevel.WARNING, Source := 'B');
fbMotionLogger.Logger(Message := 'Three', Level := E_MotionLogLevel.ERROR, Source := 'C');

logs := fbMotionLogger.GetAllMessages();

AssertTrue(
    Condition := FIND(logs, 'One') > 0 AND FIND(logs, 'Two') > 0 AND FIND(logs, 'Three') > 0,
    Message := 'GetAllMessages should include all log entries'
);
fbMotionLogger.Clear();

AssertTrue(
    Condition := fbMotionLogger.GetMessageCount() = 0,
    Message := 'Logger buffer must be empty'
);

TEST_FINISHED();
END_METHOD

END_FUNCTION_BLOCK

// ---- Test/Orchetration/FB_MotionDriveStateMachine_Test.TcPOU
FUNCTION_BLOCK FB_MotionDriveStateMachine_Test EXTENDS FB_TestSuite
VAR
    (*Test all this subject and all dependencies FB_Init call *)


    fbMotionAxisNC : ARRAY [1..20] OF FB_MotionAxisNC_TestDouble;
	stMotionCommand  : ARRAY[1..20] OF ST_MotionCommand;
    fbMotionAxisDS402 : ARRAY [1..8] OF FB_MotionAxisDS402_TestDouble;
    fbMotionLogger : ARRAY [1..20] OF FB_MotionLogger_TestDouble;
    fbMoveRequest : ARRAY [1..20] OF FB_MoveRequest_TestDouble;

END_VAR

GIvenIdlingStateIfErrorGotoErrorState_Test1();
GIvenIdlingStateIfValidatedMoveRequestThenGotoInitState_Test2();
GIvenIdlingStateAndValidatedMoveRequestIfWatchDogTImerOutThenGotoErrorState_Test3();
GivenNCAxisInitStateValidatedAbsoluteMoveRequestThenGotoStartedState_Test4();
GivenNCAxisInitStateValidatedHomeMoveRequestIfModeConfigDoneThenGotoStartedState_Test5();
GivenDS402AxisInitStateValidatedHomeMoveRequestAndNotModeConfigDoneThenLacthInitState_Test15();
GivenDS402AxisInitStateValidatedAbsoluteMoveRequestAndNotModeConfigDoneThenLatchInitState_Test17();
GivenDS402AxisInitStateValidatedHomeMoveRequestAndModeConfigDoneThenGotoStartedState_Test16();
GivenDS402AxisInitStateValidatedAbsoluteMoveRequestAndModeConfigDoneThenGotoStartedState_Test18();
GIvenStartedStatedAndErrorThenGotoErrorState_Test6();
GIvenStartedStateAndBusyStatusFromAxisThenGotoInProgressState_Test7();
GIvenStartedStateAndWatchDogTimeOutThenGotoInProgressState_Test8();
GIvenInPogressStateAndErrorThenGotoErrorState_Test9();
GivenInPogressStateAndAbortedThenGotoInterruptedState_Test10();
GIvenInPogressStateAndHomeMoveDoneStatusFromAxisThenGotoReachedState_Test11();
GIvenInPogressStateAndAbsoluteMoveDoneStatusFromAxisThenGotoReachedState_Test13();
GIvenInterruptedStateAndAbortDoneResetMoveDisablePowerThenGotoIdlingState_Test12();
GIvenReachedStateAndAxisStandStillCompleteMoveRequestThenGotoIdlingState_Test14();

METHOD PRIVATE GivenDS402AxisInitStateValidatedAbsoluteMoveRequestAndModeConfigDoneThenGotoStartedState_Test18
VAR_INST
    fbMotionDriveStateMachine : FB_MotionDriveStateMachine(
		stMotionCommand := THIS^.stMotionCommand[18],
		iMotionAxis:=THIS^.fbMotionAxisDS402[4], 
		iMoveRequest:=THIS^.fbMoveRequest[18],
		iMotionLogger := THIS^.fbMotionLogger[18]
	);
    expectedMoveState : E_MoveState := E_MoveState.STARTED;
    fbTestTimer: TON := (IN:=TRUE, PT:=T#6S);
    nTestStep : INT;
END_VAR
TEST(__POUNAME());
(*DS402 axis modeConfig did not complete within the watchDog timeout*)
CASE nTestStep OF
    0:
        fbMotionDriveStateMachine.State := E_MoveState.IDLING;
        fbMoveRequest[18].Status.bExecute := TRUE;
        fbMoveRequest[18]();
        nTestStep := nTestStep + 1;
    1:
        fbMoveRequest[18].EpicsMotorCommand := E_EpicsMotorCmd.MOVE_ABSOLUTE;
        fbMoveRequest[18]();
        fbMotionAxisDS402[4].ConfigDone := TRUE;
        fbMotionAxisDS402[4]();
        nTestStep := nTestStep + 1;
    2:
        fbMotionDriveStateMachine.State := E_MoveState.INIT;
        nTestStep := nTestStep + 1;
    3:
        AssertEquals_INT(	Expected:=expectedMoveState,
                            Actual:=fbMotionDriveStateMachine.State,
                            Message:='Drive Machine must be in STARTED state #1');
        nTestStep := nTestStep + 1;
        TEST_FINISHED();
END_CASE

fbMotionDriveStateMachine();
fbTestTimer();

IF fbTestTimer.Q THEN
    AssertTrue(Condition := FALSE, Message := CONCAT('Timed out at step: ', TO_STRING(nTestStep)));
    TEST_FINISHED();
END_IF
END_METHOD

METHOD PRIVATE GivenDS402AxisInitStateValidatedAbsoluteMoveRequestAndNotModeConfigDoneThenLatchInitState_Test17
VAR_INST
    fbMotionDriveStateMachine : FB_MotionDriveStateMachine(
		stMotionCommand := THIS^.stMotionCommand[17],
		iMotionAxis:=THIS^.fbMotionAxisDS402[3], 
		iMoveRequest:=THIS^.fbMoveRequest[17],
		iMotionLogger := THIS^.fbMotionLogger[17]
	);
    expectedMoveState : E_MoveState := E_MoveState.INIT;
    fbTestTimer: TON := (IN:=TRUE, PT:=T#6S);
    nTestStep : INT;
END_VAR
TEST(__POUNAME());
(*DS402 axis modeConfig did not complete within the watchDog timeout*)
CASE nTestStep OF
    0:
        fbMotionDriveStateMachine.State := E_MoveState.IDLING;
        fbMoveRequest[17].Status.bExecute := TRUE;
        fbMoveRequest[17]();
        nTestStep := nTestStep + 1;
    1:
        fbMoveRequest[17].EpicsMotorCommand := E_EpicsMotorCmd.MOVE_ABSOLUTE;
        fbMoveRequest[17]();
        fbMotionDriveStateMachine.State := E_MoveState.INIT;
        fbMotionDriveStateMachine();
        nTestStep := nTestStep + 1;
    2:
        AssertEquals_INT(	Expected:=expectedMoveState,
                            Actual:=fbMotionDriveStateMachine.State,
                            Message:='Drive Machine lacthes in INIT state #1');
        nTestStep := nTestStep + 1;
    3:
        IF fbMotionDriveStateMachine.WatchDogTimeOut THEN
            nTestStep := nTestStep + 1;
        END_IF
    4:
        expectedMoveState := E_MoveState.ERROR;
        AssertEquals_INT(	Expected:=expectedMoveState,
                            Actual:=fbMotionDriveStateMachine.State,
                            Message:='Drive Machine lacthes in INIT state #2');
        TEST_FINISHED();
END_CASE

fbMotionDriveStateMachine();
fbTestTimer();

IF fbTestTimer.Q THEN
    AssertTrue(Condition := FALSE, Message := CONCAT('Timed out at step: ', TO_STRING(nTestStep)));
    TEST_FINISHED();
END_IF
END_METHOD

METHOD PRIVATE GivenDS402AxisInitStateValidatedHomeMoveRequestAndModeConfigDoneThenGotoStartedState_Test16
VAR_INST
    fbMotionDriveStateMachine : FB_MotionDriveStateMachine(
		stMotionCommand := THIS^.stMotionCommand[16],
		iMotionAxis:=THIS^.fbMotionAxisDS402[2], 
		iMoveRequest:=THIS^.fbMoveRequest[16],
		iMotionLogger := THIS^.fbMotionLogger[16]
	);
    expectedMoveState : E_MoveState := E_MoveState.STARTED;
    fbTestTimer: TON := (IN:=TRUE, PT:=T#6S);
    nTestStep : INT;
END_VAR
TEST(__POUNAME());
(*DS402 axis modeConfig did not complete within the watchDog timeout*)
CASE nTestStep OF
    0:
        fbMotionDriveStateMachine.State := E_MoveState.IDLING;
        fbMoveRequest[16].Status.bExecute := TRUE;
        fbMoveRequest[16]();
        nTestStep := nTestStep + 1;
    1:
        fbMoveRequest[16].EpicsMotorCommand := E_EpicsMotorCmd.HOME;
        fbMoveRequest[16]();
        fbMotionAxisDS402[2].ConfigDone := TRUE;
        fbMotionAxisDS402[2]();
        nTestStep := nTestStep + 1;
    2:
        fbMotionDriveStateMachine.State := E_MoveState.INIT;
        nTestStep := nTestStep + 1;
    3:
        AssertEquals_INT(	Expected:=expectedMoveState,
                            Actual:=fbMotionDriveStateMachine.State,
                            Message:='Drive Machine must be in STARTED state #1');
        nTestStep := nTestStep + 1;
        TEST_FINISHED();
END_CASE

fbMotionDriveStateMachine();
fbTestTimer();

IF fbTestTimer.Q THEN
    AssertTrue(Condition := FALSE, Message := CONCAT('Timed out at step: ', TO_STRING(nTestStep)));
    TEST_FINISHED();
END_IF
END_METHOD

METHOD PRIVATE GivenDS402AxisInitStateValidatedHomeMoveRequestAndNotModeConfigDoneThenLacthInitState_Test15
VAR_INST
    fbMotionDriveStateMachine : FB_MotionDriveStateMachine(
		stMotionCommand := THIS^.stMotionCommand[15],
		iMotionAxis:=THIS^.fbMotionAxisDS402[1], 
		iMoveRequest:=THIS^.fbMoveRequest[15],
		iMotionLogger := THIS^.fbMotionLogger[15]
	);
    expectedMoveState : E_MoveState := E_MoveState.INIT;
    fbTestTimer: TON := (IN:=TRUE, PT:=T#6S);
    nTestStep : INT;
END_VAR
TEST(__POUNAME());
(*DS402 axis modeConfig did not complete within the watchDog timeout*)
CASE nTestStep OF
    0:
        fbMotionDriveStateMachine.State := E_MoveState.IDLING;
        fbMoveRequest[15].Status.bExecute := TRUE;
        fbMoveRequest[15]();
        nTestStep := nTestStep + 1;
    1:
        fbMoveRequest[15].EpicsMotorCommand := E_EpicsMotorCmd.HOME;
        fbMoveRequest[15]();
        fbMotionDriveStateMachine.State := E_MoveState.INIT;
        fbMotionDriveStateMachine();
        nTestStep := nTestStep + 1;
    2:
        AssertEquals_INT(	Expected:=expectedMoveState,
                            Actual:=fbMotionDriveStateMachine.State,
                            Message:='Drive Machine lacthes in INIT state #1');
        nTestStep := nTestStep + 1;
    3:
        IF fbMotionDriveStateMachine.WatchDogTimeOut THEN
            nTestStep := nTestStep + 1;
        END_IF
    4:
        expectedMoveState := E_MoveState.ERROR;
        AssertEquals_INT(	Expected:=expectedMoveState,
                            Actual:=fbMotionDriveStateMachine.State,
                            Message:='Drive Machine lacthes in INIT state #2');
        TEST_FINISHED();
END_CASE

fbMotionDriveStateMachine();
fbTestTimer();

IF fbTestTimer.Q THEN
    AssertTrue(Condition := FALSE, Message := CONCAT('Timed out at step: ', TO_STRING(nTestStep)));
    TEST_FINISHED();
END_IF
END_METHOD

METHOD PRIVATE GIvenIdlingStateAndValidatedMoveRequestIfWatchDogTImerOutThenGotoErrorState_Test3
VAR_INST
    fbMotionDriveStateMachine : FB_MotionDriveStateMachine(
		stMotionCommand := THIS^.stMotionCommand[3],
		iMotionAxis:=THIS^.fbMotionAxisNC[3], 
		iMoveRequest:=THIS^.fbMoveRequest[3],
		iMotionLogger := THIS^.fbMotionLogger[3]
	);
    expectedMoveState : E_MoveState := E_MoveState.ERROR;
    fbTestTimer: TON := (IN:=TRUE, PT:=T#6S);
    nTestStep : INT;
END_VAR
TEST(__POUNAME());
CASE nTestStep OF
    0:
        fbMotionDriveStateMachine.State := E_MoveState.IDLING;
        fbMoveRequest[3].Status.bExecute := TRUE;
        fbMoveRequest[3]();
        fbMotionDriveStateMachine();
        nTestStep := nTestStep + 1;
    1:
        IF fbMotionDriveStateMachine.WatchDogStatus THEN
            nTestStep := nTestStep + 1;
        END_IF

    2:
        IF fbMotionDriveStateMachine.WatchDogTimeOut THEN
            nTestStep := nTestStep + 1;
        END_IF
    3:
        AssertEquals_INT(	Expected:=expectedMoveState,
                            Actual:=fbMotionDriveStateMachine.State,
                            Message:='Drive Machine state must be ERROR #1');
        AssertTrue(Condition := fbMotionDriveStateMachine.Error, Message := 'Motion Drive state machine must be in error state #2');
        nTestStep := nTestStep + 1;
        TEST_FINISHED();
END_CASE

fbMotionDriveStateMachine();
fbTestTimer();

IF fbTestTimer.Q THEN
    AssertTrue(Condition := FALSE, Message := CONCAT('Timed out at step: ', TO_STRING(nTestStep)));
    TEST_FINISHED();
END_IF
END_METHOD

METHOD PRIVATE GIvenIdlingStateIfErrorGotoErrorState_Test1
VAR_INST
    fbMotionDriveStateMachine : FB_MotionDriveStateMachine(
		stMotionCommand := THIS^.stMotionCommand[1],
		iMotionAxis:=THIS^.fbMotionAxisNC[1], 
		iMoveRequest:=THIS^.fbMoveRequest[1],
		iMotionLogger := THIS^.fbMotionLogger[1]
	);
    expectedMoveState : E_MoveState := E_MoveState.ERROR;
END_VAR
TEST(__POUNAME());

fbMotionDriveStateMachine.State := E_MoveState.IDLING;
fbMotionDriveStateMachine.StateMachine(Error:=TRUE);
fbMotionDriveStateMachine();
AssertEquals_INT(	Expected:=expectedMoveState,
                    Actual:=fbMotionDriveStateMachine.State,
                    Message:='Drive Machine state must be ERROR #1');


TEST_FINISHED();
END_METHOD

METHOD PRIVATE GIvenIdlingStateIfValidatedMoveRequestThenGotoInitState_Test2
VAR_INST
    fbMotionDriveStateMachine : FB_MotionDriveStateMachine(
		stMotionCommand := THIS^.stMotionCommand[2],
		iMotionAxis:=THIS^.fbMotionAxisNC[2], 
		iMoveRequest:=THIS^.fbMoveRequest[2],
		iMotionLogger := THIS^.fbMotionLogger[2]
	);
    expectedMoveState : E_MoveState := E_MoveState.INIT;
END_VAR
TEST(__POUNAME());

fbMotionDriveStateMachine.State := E_MoveState.IDLING;
fbMoveRequest[2].Status.bExecute := TRUE;
fbMoveRequest[2]();
fbMotionDriveStateMachine();

AssertEquals_INT(	Expected:=expectedMoveState,
                    Actual:=fbMotionDriveStateMachine.State,
                    Message:='Drive Machine state must be INIT #1');

AssertTrue(Condition := THIS^.fbMoveRequest[2].Status.bExecute, Message := 'Move must be validated #2');

TEST_FINISHED();
END_METHOD

METHOD PRIVATE GivenInPogressStateAndAbortedThenGotoInterruptedState_Test10
VAR_INST
    fbMotionDriveStateMachine : FB_MotionDriveStateMachine(
		stMotionCommand := THIS^.stMotionCommand[10],
		iMotionAxis:=THIS^.fbMotionAxisNC[10], 
		iMoveRequest:=THIS^.fbMoveRequest[10],
		iMotionLogger := THIS^.fbMotionLogger[10]
	);
    expectedMoveState : E_MoveState := E_MoveState.INTERRUPTED;
END_VAR
TEST(__POUNAME());

fbMotionAxisNC[10].Status.bAborted := TRUE;
fbMotionAxisNC[10]();
fbMotionDriveStateMachine.State := E_MoveState.IN_PROGRESS;
fbMotionDriveStateMachine();
AssertEquals_INT(	Expected:=expectedMoveState,
                    Actual:=fbMotionDriveStateMachine.State,
                    Message:='Drive must be in INTERRUPTED state #1');


TEST_FINISHED();
END_METHOD

METHOD PRIVATE GIvenInPogressStateAndAbsoluteMoveDoneStatusFromAxisThenGotoReachedState_Test13
VAR_INST
    fbMotionDriveStateMachine : FB_MotionDriveStateMachine(
		stMotionCommand := THIS^.stMotionCommand[13],
		iMotionAxis:=THIS^.fbMotionAxisNC[13], 
		iMoveRequest:=THIS^.fbMoveRequest[13],
		iMotionLogger := THIS^.fbMotionLogger[13]
	);
    expectedMoveState : E_MoveState := E_MoveState.REACHED;
END_VAR
TEST(__POUNAME());

fbMotionAxisNC[13].Status.bMoveAbsoluteDone := TRUE;
fbMotionAxisNC[13]();
fbMotionDriveStateMachine.State := E_MoveState.IN_PROGRESS;
fbMotionDriveStateMachine();
AssertEquals_INT(	Expected:=expectedMoveState,
                    Actual:=fbMotionDriveStateMachine.State,
                    Message:='Drive must be in REACHED state #1');


TEST_FINISHED();
END_METHOD

METHOD PRIVATE GIvenInPogressStateAndErrorThenGotoErrorState_Test9
VAR_INST
    fbMotionDriveStateMachine : FB_MotionDriveStateMachine(
		stMotionCommand := THIS^.stMotionCommand[9],
		iMotionAxis:=THIS^.fbMotionAxisNC[9], 
		iMoveRequest:=THIS^.fbMoveRequest[9],
		iMotionLogger := THIS^.fbMotionLogger[9]
	);
    expectedMoveState : E_MoveState := E_MoveState.ERROR;
END_VAR
TEST(__POUNAME());

fbMotionDriveStateMachine.State := E_MoveState.IN_PROGRESS;
fbMotionDriveStateMachine.StateMachine(Error:=TRUE);
fbMotionDriveStateMachine();

AssertEquals_INT(	Expected:=expectedMoveState,
                    Actual:=fbMotionDriveStateMachine.State,
                    Message:='Drive Machine state must be ERROR #1');

TEST_FINISHED();
END_METHOD

METHOD PRIVATE GIvenInPogressStateAndHomeMoveDoneStatusFromAxisThenGotoReachedState_Test11
VAR_INST
    fbMotionDriveStateMachine : FB_MotionDriveStateMachine(
		stMotionCommand := THIS^.stMotionCommand[11],
		iMotionAxis:=THIS^.fbMotionAxisNC[11], 
		iMoveRequest:=THIS^.fbMoveRequest[11],
		iMotionLogger := THIS^.fbMotionLogger[11]
	);
    expectedMoveState : E_MoveState := E_MoveState.REACHED;
END_VAR
TEST(__POUNAME());

fbMotionAxisNC[11].Status.bHomeDone := TRUE;
fbMotionAxisNC[11]();
fbMotionDriveStateMachine.State := E_MoveState.IN_PROGRESS;
fbMotionDriveStateMachine();
AssertEquals_INT(	Expected:=expectedMoveState,
                    Actual:=fbMotionDriveStateMachine.State,
                    Message:='Drive must be in REACHED state #1');


TEST_FINISHED();
END_METHOD

METHOD PRIVATE GIvenInterruptedStateAndAbortDoneResetMoveDisablePowerThenGotoIdlingState_Test12
VAR_INST
    fbMotionDriveStateMachine : FB_MotionDriveStateMachine(
		stMotionCommand := THIS^.stMotionCommand[12],
		iMotionAxis:=THIS^.fbMotionAxisNC[12], 
		iMoveRequest:=THIS^.fbMoveRequest[12],
		iMotionLogger := THIS^.fbMotionLogger[12]
	);	
    expectedMoveState : E_MoveState := E_MoveState.IDLING;
    fbTestTimer: TON := (IN:=TRUE, PT:=T#2S);
    nTestStep : INT;
END_VAR
TEST(__POUNAME());
CASE 	nTestStep OF
    0:
        fbMotionAxisNC[12].Status.bAborted := TRUE;
        fbMotionDriveStateMachine.State := E_MoveState.IN_PROGRESS;
        nTestStep := nTestStep + 1;
    1:
        // now we should be in the interrupted state
        fbMotionAxisNC[12].Status.bAbortDone := TRUE;
        fbMotionAxisNC[12]();
        nTestStep := nTestStep + 1;
END_CASE

fbMotionAxisNC[12]();
fbMotionDriveStateMachine();
fbTestTimer();

IF nTestStep = 2 THEN
    AssertEquals_INT(	Expected:=expectedMoveState,
                    Actual:=fbMotionDriveStateMachine.State,
                    Message:='Drive must be in IDLING state #1');
    TEST_FINISHED();
ELSIF fbTestTimer.Q THEN
    AssertTrue(Condition := FALSE, Message := CONCAT('Timed out at step: ', TO_STRING(nTestStep)));
    TEST_FINISHED();
END_IF
END_METHOD

METHOD PRIVATE GivenNCAxisInitStateValidatedAbsoluteMoveRequestThenGotoStartedState_Test4
VAR_INST
    fbMotionDriveStateMachine : FB_MotionDriveStateMachine(
		stMotionCommand := THIS^.stMotionCommand[4],
		iMotionAxis:=THIS^.fbMotionAxisNC[4], 
		iMoveRequest:=THIS^.fbMoveRequest[4],
		iMotionLogger := THIS^.fbMotionLogger[4]
	);
    expectedMoveState : E_MoveState := E_MoveState.STARTED;
END_VAR
TEST(__POUNAME());

fbMoveRequest[4].EpicsMotorCommand := E_EpicsMotorCmd.MOVE_ABSOLUTE;
fbMoveRequest[4]();
fbMotionDriveStateMachine.State := E_MoveState.INIT;
fbMotionDriveStateMachine();


expectedMoveState := E_MoveState.STARTED;
AssertEquals_INT(	Expected:=expectedMoveState,
                    Actual:=fbMotionDriveStateMachine.State,
                    Message:='Drive Machine state must be STARTED #1');
TEST_FINISHED();
END_METHOD

METHOD PRIVATE GivenNCAxisInitStateValidatedHomeMoveRequestIfModeConfigDoneThenGotoStartedState_Test5
VAR_INST
    fbMotionDriveStateMachine : FB_MotionDriveStateMachine(
		stMotionCommand := THIS^.stMotionCommand[5],
		iMotionAxis:=THIS^.fbMotionAxisNC[5], 
		iMoveRequest:=THIS^.fbMoveRequest[5],
		iMotionLogger := THIS^.fbMotionLogger[5]
	);
    expectedMoveState : E_MoveState := E_MoveState.ERROR;
    nTestStep : INT;
END_VAR
TEST(__POUNAME());

fbMoveRequest[5].EpicsMotorCommand := E_EpicsMotorCmd.HOME;
fbMoveRequest[5]();
fbMotionDriveStateMachine.State := E_MoveState.INIT;
fbMotionDriveStateMachine();


expectedMoveState := E_MoveState.STARTED;
AssertEquals_INT(	Expected:=expectedMoveState,
                    Actual:=fbMotionDriveStateMachine.State,
                    Message:='Drive Machine state must be STARTED #1');
TEST_FINISHED();
END_METHOD

METHOD PRIVATE GIvenReachedStateAndAxisStandStillCompleteMoveRequestThenGotoIdlingState_Test14
VAR_INST
    fbMotionDriveStateMachine : FB_MotionDriveStateMachine(
		stMotionCommand := THIS^.stMotionCommand[14],
		iMotionAxis:=THIS^.fbMotionAxisNC[14], 
		iMoveRequest:=THIS^.fbMoveRequest[14],
		iMotionLogger := THIS^.fbMotionLogger[14]
	);
    expectedMoveState : E_MoveState := E_MoveState.IDLING;
END_VAR
TEST(__POUNAME());

fbMotionAxisNC[14].Status.bStandStill := TRUE;
fbMotionAxisNC[14].Status.bHomeDone := FALSE;
fbMotionAxisNC[14].Status.bMoveAbsoluteDone := TRUE;
fbMotionAxisNC[14]();
fbMotionDriveStateMachine.State := E_MoveState.REACHED;
fbMotionDriveStateMachine();

AssertEquals_INT(	Expected:=expectedMoveState,
                    Actual:=fbMotionDriveStateMachine.State,
                    Message:='Drive must be in IDLING state #1');


TEST_FINISHED();
END_METHOD

METHOD PRIVATE GIvenStartedStateAndBusyStatusFromAxisThenGotoInProgressState_Test7
VAR_INST
    fbMotionDriveStateMachine : FB_MotionDriveStateMachine(
		stMotionCommand := THIS^.stMotionCommand[7],
		iMotionAxis:=THIS^.fbMotionAxisNC[7], 
		iMoveRequest:=THIS^.fbMoveRequest[7],
		iMotionLogger := THIS^.fbMotionLogger[7]
	);
    expectedMoveState : E_MoveState := E_MoveState.IN_PROGRESS;
    nTestStep : INT;
END_VAR
TEST(__POUNAME());
CASE nTestStep OF
    0:
        fbMotionDriveStateMachine.State := E_MoveState.STARTED;
        fbMotionAxisNC[7].Status.bBusy := TRUE;
        nTestStep := nTestStep + 1;
    1:
        AssertEquals_INT(	Expected:=expectedMoveState,
                            Actual:=fbMotionDriveStateMachine.State,
                            Message:='Drive Machine must be IN_PROGRESS state #1');
        TEST_FINISHED();
END_CASE

fbMotionDriveStateMachine();
END_METHOD

METHOD PRIVATE GIvenStartedStateAndWatchDogTimeOutThenGotoInProgressState_Test8
VAR_INST
    fbMotionDriveStateMachine : FB_MotionDriveStateMachine(
		stMotionCommand := THIS^.stMotionCommand[8],
		iMotionAxis:=THIS^.fbMotionAxisNC[8], 
		iMoveRequest:=THIS^.fbMoveRequest[8],
		iMotionLogger := THIS^.fbMotionLogger[8]
	);
    expectedMoveState : E_MoveState := E_MoveState.ERROR;
    fbTestTimer: TON := (IN:=TRUE, PT:=T#6S);
    nTestStep : INT;
END_VAR
TEST(__POUNAME());
CASE nTestStep OF
    0:
        fbMoveRequest[8].Status.bExecute := TRUE;
        fbMoveRequest[8]();
        fbMotionDriveStateMachine.State := E_MoveState.STARTED;
        fbMotionDriveStateMachine.WatchDog := TRUE;
        fbMotionDriveStateMachine();
        nTestStep := nTestStep + 1;
    1:
        IF fbMotionDriveStateMachine.WatchDogStatus THEN
            nTestStep := nTestStep + 1;
        END_IF

